  MoveL 1864 to (-16.69, 20.93, 85) mm, rotated rx 180 ry 0 rz -180 deg; joints [-156.025, -53.771, -94.051, 27.718, 60.883, -14.341]
  Call Extruder(17898.90608)
  MoveL 1865 to (-20.93, 16.69, 85) mm, rotated rx -180 ry 0 rz -180 deg; joints [-156.374, -53.467, -95.005, 27.167, 61.375, -13.813]
  Call Extruder(17908.27099)
  MoveL 1866 to (-24.11, 11.61, 85) mm, rotated rx -180 ry 0 rz 180 deg; joints [-156.928, -53.206, -95.842, 26.413, 61.758, -13.226]
  Call Extruder(17917.63579)
  MoveL 1867 to (-26.09, 5.96, 85) mm, rotated rx -180 ry 0 rz -180 deg; joints [-157.665, -52.998, -96.517, 25.49, 62.014, -12.61]
  Call Extruder(17927.00089)
  MoveL 1868 to (-26.77, 0, 85) mm, rotated rx 180 ry 0 rz -180 deg; joints [-158.546, -52.854, -96.993, 24.441, 62.127, -11.995]
  Call Extruder(17931.78963)
  MoveL 1869 to (-26.42, -3.05, 85) mm, rotated rx 180 ry 0 rz -180 deg; joints [-159.044, -52.814, -97.124, 23.87, 62.108, -11.695]
  Set speed (130.0 mm/s)
  MoveL 1870 to (-41.86, -6.3, 85) mm, rotated rx -180 ry 0 rz 180 deg; joints [-158.606, -52.066, -99.698, 23.975, 63.864, -11.084]
  Call Extruder(17936.78748)
  Set speed (60.0 mm/s)
  MoveL 1871 to (-41.51, -9.47, 85) mm, rotated rx -180 ry 0 rz 180 deg; joints [-159.151, -52.029, -99.83, 23.359, 63.847, -10.778]
  Call Extruder(17951.68313)
  MoveL 1872 to (-38.36, -18.47, 85) mm, rotated rx 180 ry 0 rz 180 deg; joints [-160.835, -52.023, -99.85, 21.508, 63.558, -9.953]
  Call Extruder(17966.57898)
  MoveL 1873 to (-33.28, -26.54, 85) mm, rotated rx 180 ry 0 rz 180 deg; joints [-162.466, -52.128, -99.478, 19.757, 63.035, -9.25]
  Call Extruder(17981.47480)
  MoveL 1874 to (-26.54, -33.28, 85) mm, rotated rx 180 ry 0 rz -180 deg; joints [-163.93, -52.339, -98.738, 18.218, 62.307, -8.696]
  Call Extruder(17996.37065)
  MoveL 1875 to (-18.47, -38.36, 85) mm, rotated rx 180 ry 0 rz 180 deg; joints [-165.137, -52.65, -97.673, 16.986, 61.41, -8.316]
  Call Extruder(18011.26630)
  MoveL 1876 to (-9.47, -41.51, 85) mm, rotated rx -180 ry 0 rz 180 deg; joints [-166.024, -53.05, -96.347, 16.127, 60.395, -8.129]
  Call Extruder(18026.16218)
  MoveL 1877 to (0, -42.57, 85) mm, rotated rx -180 ry 0 rz 180 deg; joints [-166.562, -53.521, -94.833, 15.678, 59.317, -8.151]
  Call Extruder(18033.93795)
  MoveL 1878 to (4.95, -42.02, 85) mm, rotated rx 180 ry 0 rz 180 deg; joints [-166.659, -53.791, -93.99, 15.659, 58.75, -8.274]
  Call Extruder(18041.05804)
  MoveL 1879 to (9.47, -41.51, 85) mm, rotated rx -180 ry 0 rz 180 deg; joints [-166.745, -54.043, -93.212, 15.646, 58.231, -8.388]
  Call Extruder(18055.95371)
  MoveL 1880 to (18.47, -38.36, 85) mm, rotated rx -180 ry 0 rz 180 deg; joints [-166.591, -54.589, -91.565, 16.015, 57.195, -8.839]
  Call Extruder(18070.84955)
  MoveL 1881 to (26.54, -33.29, 85) mm, rotated rx 180 ry 0 rz 180 deg; joints [-166.133, -55.132, -89.973, 16.751, 56.262, -9.49]
  Call Extruder(18085.74538)
  MoveL 1882 to (33.29, -26.54, 85) mm, rotated rx 180 ry 0 rz 180 deg; joints [-165.409, -55.642, -88.512, 17.803, 55.478, -10.315]
  Call Extruder(18100.64123)
  MoveL 1883 to (38.36, -18.47, 85) mm, rotated rx -180 ry 0 rz 180 deg; joints [-164.468, -56.091, -87.25, 19.109, 54.883, -11.272]
  Call Extruder(18115.53688)
  MoveL 1884 to (41.5, -9.47, 85) mm, rotated rx 180 ry 0 rz 180 deg; joints [-163.355, -56.454, -86.244, 20.599, 54.506, -12.31]
  Call Extruder(18130.43275)
  MoveL 1885 to (42.57, 0, 85) mm, rotated rx 180 ry 0 rz 180 deg; joints [-162.12, -56.711, -85.541, 22.195, 54.365, -13.372]
  Call Extruder(18145.32862)
  MoveL 1886 to (41.51, 9.47, 85) mm, rotated rx -180 ry 0 rz 180 deg; joints [-160.81, -56.847, -85.172, 23.824, 54.464, -14.393]
  Call Extruder(18160.22429)
  MoveL 1887 to (38.36, 18.47, 85) mm, rotated rx 180 ry 0 rz 180 deg; joints [-159.475, -56.853, -85.155, 25.41, 54.797, -15.316]
  Call Extruder(18175.12013)
  MoveL 1888 to (33.29, 26.54, 85) mm, rotated rx 180 ry 0 rz 180 deg; joints [-158.16, -56.73, -85.489, 26.888, 55.342, -16.085]
  Call Extruder(18190.01595)
  MoveL 1889 to (26.54, 33.28, 85) mm, rotated rx 180 ry 0 rz 180 deg; joints [-156.916, -56.485, -86.16, 28.2, 56.071, -16.662]
  Call Extruder(18204.91180)
  MoveL 1890 to (18.47, 38.36, 85) mm, rotated rx 180 ry 0 rz -180 deg; joints [-155.789, -56.131, -87.138, 29.294, 56.944, -17.016]
  Call Extruder(18219.80746)
  MoveL 1891 to (9.47, 41.51, 85) mm, rotated rx 180 ry 0 rz 180 deg; joints [-154.828, -55.689, -88.377, 30.132, 57.919, -17.133]
  Call Extruder(18234.70334)
  MoveL 1892 to (0, 42.57, 85) mm, rotated rx 180 ry 0 rz 180 deg; joints [-154.081, -55.184, -89.821, 30.678, 58.948, -17.014]
  Call Extruder(18249.59921)
  MoveL 1893 to (-9.47, 41.51, 85) mm, rotated rx 180 ry 0 rz 180 deg; joints [-153.594, -54.644, -91.403, 30.905, 59.984, -16.67]
  Call Extruder(18264.49486)
  MoveL 1894 to (-18.47, 38.36, 85) mm, rotated rx 180 ry 0 rz -180 deg; joints [-153.408, -54.096, -93.048, 30.791, 60.979, -16.124]
  Call Extruder(18279.39071)
  MoveL 1895 to (-26.54, 33.29, 85) mm, rotated rx 180 ry 0 rz 180 deg; joints [-153.557, -53.571, -94.676, 30.322, 61.888, -15.408]
  Call Extruder(18294.28653)
  MoveL 1896 to (-33.28, 26.54, 85) mm, rotated rx 180 ry 0 rz 180 deg; joints [-154.059, -53.094, -96.204, 29.499, 62.669, -14.561]
  Call Extruder(18309.18238)
  MoveL 1897 to (-38.36, 18.47, 85) mm, rotated rx 180 ry 0 rz -180 deg; joints [-154.913, -52.686, -97.552, 28.338, 63.284, -13.628]
  Call Extruder(18324.07804)
  MoveL 1898 to (-41.5, 9.47, 85) mm, rotated rx -180 ry 0 rz 180 deg; joints [-156.091, -52.366, -98.646, 26.877, 63.701, -12.656]
  Call Extruder(18338.97391)
  MoveL 1899 to (-42.57, 0, 85) mm, rotated rx 180 ry 0 rz -180 deg; joints [-157.533, -52.144, -99.421, 25.187, 63.894, -11.692]
  Call Extruder(18346.52819)
  MoveL 1900 to (-42.03, -4.8, 85) mm, rotated rx 180 ry 0 rz 180 deg; joints [-158.35, -52.084, -99.634, 24.263, 63.871, -11.227]
  Set speed (130.0 mm/s)
  MoveL 1901 to (-54.1, -7.67, 85) mm, rotated rx 180 ry 0 rz 180 deg; joints [-158.024, -51.54, -101.626, 24.334, 65.254, -10.72]
  Call Extruder(18350.60082)
  Set speed (30.0 mm/s)
  MoveL 1902 to (-53.59, -12.23, 85) mm, rotated rx 180 ry 0 rz -180 deg; joints [-158.835, -51.49, -101.819, 23.429, 65.236, -10.288]
  Call Extruder(18361.53095)
  MoveL 1903 to (-49.52, -23.85, 85) mm, rotated rx 180 ry 0 rz 180 deg; joints [-161.095, -51.483, -101.845, 20.97, 64.87, -9.244]
  Call Extruder(18372.46124)
  MoveL 1904 to (-42.98, -34.27, 85) mm, rotated rx -180 ry 0 rz 180 deg; joints [-163.275, -51.612, -101.354, 18.642, 64.197, -8.354]
  Call Extruder(18383.39136)
  MoveL 1905 to (-34.27, -42.98, 85) mm, rotated rx 180 ry 0 rz 180 deg; joints [-165.21, -51.876, -100.38, 16.611, 63.25, -7.647]
  Call Extruder(18394.32164)
  MoveL 1906 to (-23.85, -49.53, 85) mm, rotated rx 180 ry 0 rz 180 deg; joints [-166.774, -52.268, -98.985, 15.006, 62.083, -7.154]
  Call Extruder(18405.25177)
  MoveL 1907 to (-12.23, -53.59, 85) mm, rotated rx -180 ry 0 rz 180 deg; joints [-167.889, -52.775, -97.254, 13.913, 60.762, -6.899]
  Call Extruder(18416.18200)
  MoveL 1908 to (0, -54.97, 85) mm, rotated rx -180 ry 0 rz 180 deg; joints [-168.526, -53.378, -95.288, 13.367, 59.36, -6.905]
  Call Extruder(18421.83349)
  MoveL 1909 to (6.32, -54.26, 85) mm, rotated rx 180 ry 0 rz 180 deg; joints [-168.616, -53.721, -94.208, 13.366, 58.632, -7.051]
  Call Extruder(18427.11222)
  MoveL 1910 to (12.23, -53.59, 85) mm, rotated rx -180 ry 0 rz 180 deg; joints [-168.697, -54.05, -93.19, 13.37, 57.952, -7.188]
  Call Extruder(18438.04236)
  MoveL 1911 to (23.85, -49.53, 85) mm, rotated rx 180 ry 0 rz 180 deg; joints [-168.436, -54.757, -91.068, 13.891, 56.611, -7.75]
  Call Extruder(18448.97264)
  MoveL 1912 to (34.27, -42.98, 85) mm, rotated rx 180 ry 0 rz 180 deg; joints [-167.797, -55.462, -89.022, 14.879, 55.403, -8.579]
  Call Extruder(18459.90276)
  MoveL 1913 to (42.98, -34.27, 85) mm, rotated rx -180 ry 0 rz 180 deg; joints [-166.837, -56.127, -87.148, 16.266, 54.391, -9.642]
  Call Extruder(18470.83304)
  MoveL 1914 to (49.53, -23.85, 85) mm, rotated rx -180 ry 0 rz 180 deg; joints [-165.618, -56.714, -85.531, 17.968, 53.624, -10.888]
  Call Extruder(18481.76317)
  MoveL 1915 to (53.59, -12.23, 85) mm, rotated rx 180 ry 0 rz -180 deg; joints [-164.2, -57.19, -84.244, 19.895, 53.141, -12.248]
  Call Extruder(18492.69340)
  MoveL 1916 to (54.97, 0, 85) mm, rotated rx 180 ry 0 rz 180 deg; joints [-162.641, -57.527, -83.344, 21.948, 52.964, -13.643]
  Call Extruder(18503.62362)
  MoveL 1917 to (53.59, 12.23, 85) mm, rotated rx 180 ry 0 rz 180 deg; joints [-160.996, -57.705, -82.872, 24.029, 53.1, -14.986]
  Call Extruder(18514.55376)
  MoveL 1918 to (49.52, 23.85, 85) mm, rotated rx -180 ry 0 rz -180 deg; joints [-159.322, -57.714, -82.85, 26.044, 53.537, -16.195]
  Call Extruder(18525.48404)
  MoveL 1919 to (42.98, 34.27, 85) mm, rotated rx -180 ry 0 rz 180 deg; joints [-157.673, -57.552, -83.278, 27.912, 54.249, -17.198]
  Call Extruder(18536.41416)
  MoveL 1920 to (34.27, 42.98, 85) mm, rotated rx -180 ry 0 rz 180 deg; joints [-156.102, -57.23, -84.137, 29.563, 55.194, -17.94]
  Call Extruder(18547.34444)
  MoveL 1921 to (23.85, 49.52, 85) mm, rotated rx -180 ry 0 rz 180 deg; joints [-154.667, -56.767, -85.388, 30.942, 56.322, -18.388]
  Call Extruder(18558.27458)
  MoveL 1922 to (12.23, 53.59, 85) mm, rotated rx 180 ry 0 rz 180 deg; joints [-153.426, -56.19, -86.975, 32.004, 57.576, -18.526]
  Call Extruder(18569.20480)
  MoveL 1923 to (0, 54.97, 85) mm, rotated rx -180 ry 0 rz 180 deg; joints [-152.438, -55.531, -88.827, 32.711, 58.896, -18.355]
  Call Extruder(18580.13502)
  MoveL 1924 to (-12.23, 53.59, 85) mm, rotated rx 180 ry 0 rz 180 deg; joints [-151.764, -54.828, -90.86, 33.03, 60.223, -17.894]
  Call Extruder(18591.06516)
  MoveL 1925 to (-23.85, 49.52, 85) mm, rotated rx 180 ry 0 rz 180 deg; joints [-151.463, -54.119, -92.979, 32.93, 61.497, -17.175]
  Call Extruder(18601.99544)
  MoveL 1926 to (-34.27, 42.98, 85) mm, rotated rx 180 ry 0 rz 180 deg; joints [-151.589, -53.442, -95.084, 32.385, 62.663, -16.239]
  Call Extruder(18612.92556)
  MoveL 1927 to (-42.98, 34.27, 85) mm, rotated rx 180 ry 0 rz -180 deg; joints [-152.179, -52.831, -97.068, 31.381, 63.669, -15.139]
  Call Extruder(18623.85584)
  MoveL 1928 to (-49.52, 23.85, 85) mm, rotated rx 180 ry 0 rz 180 deg; joints [-153.248, -52.313, -98.827, 29.924, 64.469, -13.933]
  Call Extruder(18634.78598)
  MoveL 1929 to (-53.59, 12.23, 85) mm, rotated rx 180 ry 0 rz 180 deg; joints [-154.769, -51.91, -100.259, 28.051, 65.018, -12.683]
  Call Extruder(18645.71620)
  MoveL 1930 to (-54.97, 0, 85) mm, rotated rx 180 ry 0 rz -180 deg; joints [-156.673, -51.633, -101.278, 25.844, 65.282, -11.45]
  Call Extruder(18651.24182)
  MoveL 1931 to (-54.27, -6.18, 85) mm, rotated rx 180 ry 0 rz -180 deg; joints [-157.76, -51.558, -101.561, 24.629, 65.26, -10.861]
  Set speed (130.0 mm/s)
  MoveL 1932 to (-49.9, -9.51, 85) mm, rotated rx -180 ry 0 rz 180 deg; joints [-158.616, -51.679, -101.105, 23.764, 64.795, -10.62]
  MoveL 1933 to (1.69, -13.14, 85) mm, rotated rx 180 ry 0 rz -180 deg; joints [-162.112, -54.05, -93.191, 20.997, 59.006, -11.18]
  Call Extruder(18653.24626)
  Set speed (80.0 mm/s)
  MoveL 1934 to (2.97, -12.99, 85) mm, rotated rx -180 ry 0 rz -180 deg; joints [-162.152, -54.121, -92.974, 20.982, 58.862, -11.217]
  Call Extruder(18657.90984)
  MoveL 1935 to (5.78, -12.01, 85) mm, rotated rx 180 ry 0 rz -180 deg; joints [-162.141, -54.291, -92.457, 21.071, 58.541, -11.37]
  Call Extruder(18662.57346)
  MoveL 1936 to (8.31, -10.42, 85) mm, rotated rx -180 ry 0 rz -180 deg; joints [-162.027, -54.459, -91.954, 21.277, 58.25, -11.581]
  Call Extruder(18667.23766)
  MoveL 1937 to (10.42, -8.31, 85) mm, rotated rx 180 ry 0 rz -180 deg; joints [-161.819, -54.615, -91.489, 21.587, 58.005, -11.84]
  Call Extruder(18671.90129)
  MoveL 1938 to (12.01, -5.78, 85) mm, rotated rx -180 ry 0 rz 180 deg; joints [-161.529, -54.751, -91.086, 21.984, 57.817, -12.135]
  Call Extruder(18676.56485)
  MoveL 1939 to (12.99, -2.97, 85) mm, rotated rx -180 ry 0 rz -180 deg; joints [-161.171, -54.861, -90.763, 22.448, 57.696, -12.451]
  Call Extruder(18681.22881)
  MoveL 1940 to (13.33, 0, 85) mm, rotated rx 180 ry 0 rz -180 deg; joints [-160.763, -54.938, -90.537, 22.956, 57.648, -12.771]
  Call Extruder(18685.89276)
  MoveL 1941 to (12.99, 2.97, 85) mm, rotated rx 180 ry 0 rz 180 deg; joints [-160.324, -54.979, -90.418, 23.482, 57.674, -13.078]
  Call Extruder(18690.55633)
  MoveL 1942 to (12.01, 5.78, 85) mm, rotated rx -180 ry 0 rz -180 deg; joints [-159.874, -54.981, -90.412, 24.001, 57.774, -13.357]
  Call Extruder(18695.21996)
  MoveL 1943 to (10.42, 8.31, 85) mm, rotated rx -180 ry 0 rz 180 deg; joints [-159.432, -54.944, -90.52, 24.489, 57.941, -13.592]
  Call Extruder(18699.88415)
  MoveL 1944 to (8.31, 10.42, 85) mm, rotated rx 180 ry 0 rz 180 deg; joints [-159.021, -54.87, -90.736, 24.924, 58.168, -13.771]
  Call Extruder(18704.54778)
  MoveL 1945 to (5.78, 12.01, 85) mm, rotated rx 180 ry 0 rz -180 deg; joints [-158.657, -54.763, -91.05, 25.285, 58.442, -13.886]
  Call Extruder(18709.21134)
  MoveL 1946 to (2.97, 12.99, 85) mm, rotated rx -180 ry 0 rz 180 deg; joints [-158.359, -54.629, -91.446, 25.555, 58.75, -13.931]
  Call Extruder(18713.87530)
  MoveL 1947 to (0, 13.33, 85) mm, rotated rx 180 ry 0 rz 180 deg; joints [-158.143, -54.475, -91.906, 25.72, 59.078, -13.903]
  Call Extruder(18718.53925)
  MoveL 1948 to (-2.97, 13, 85) mm, rotated rx 180 ry 0 rz 180 deg; joints [-158.019, -54.308, -92.406, 25.774, 59.408, -13.806]
  Call Extruder(18723.20282)
  MoveL 1949 to (-5.78, 12.01, 85) mm, rotated rx 180 ry 0 rz 180 deg; joints [-157.997, -54.138, -92.923, 25.71, 59.725, -13.644]
  Call Extruder(18727.86645)
  MoveL 1950 to (-8.31, 10.42, 85) mm, rotated rx 180 ry 0 rz 180 deg; joints [-158.08, -53.972, -93.43, 25.531, 60.013, -13.427]
  Call Extruder(18732.53064)
  MoveL 1951 to (-10.42, 8.31, 85) mm, rotated rx 180 ry 0 rz 180 deg; joints [-158.266, -53.819, -93.901, 25.244, 60.259, -13.165]
  Call Extruder(18737.19427)
  MoveL 1952 to (-12.01, 5.78, 85) mm, rotated rx -180 ry 0 rz 180 deg; joints [-158.549, -53.687, -94.314, 24.86, 60.448, -12.872]
  Call Extruder(18741.85784)
  MoveL 1953 to (-12.99, 2.97, 85) mm, rotated rx -180 ry 0 rz -180 deg; joints [-158.913, -53.581, -94.645, 24.398, 60.573, -12.563]
  Call Extruder(18746.52180)
  MoveL 1954 to (-13.33, 0, 85) mm, rotated rx 180 ry 0 rz 180 deg; joints [-159.341, -53.507, -94.878, 23.881, 60.627, -12.253]
  Call Extruder(18751.18574)
  MoveL 1955 to (-12.99, -2.97, 85) mm, rotated rx 180 ry 0 rz 180 deg; joints [-159.811, -53.468, -95.001, 23.336, 60.605, -11.956]
  Call Extruder(18755.84931)
  MoveL 1956 to (-12.01, -5.78, 85) mm, rotated rx 180 ry 0 rz 180 deg; joints [-160.294, -53.467, -95.007, 22.791, 60.51, -11.687]
  Call Extruder(18760.51294)
  MoveL 1957 to (-10.42, -8.31, 85) mm, rotated rx 180 ry 0 rz 180 deg; joints [-160.766, -53.502, -94.895, 22.276, 60.345, -11.458]
  Call Extruder(18765.17714)
  MoveL 1958 to (-8.31, -10.42, 85) mm, rotated rx -180 ry 0 rz 180 deg; joints [-161.2, -53.572, -94.673, 21.819, 60.118, -11.281]
  Call Extruder(18769.84076)
  MoveL 1959 to (-5.78, -12.01, 85) mm, rotated rx 180 ry 0 rz 180 deg; joints [-161.572, -53.675, -94.35, 21.445, 59.842, -11.163]
  Call Extruder(18774.50433)
  MoveL 1960 to (-2.97, -12.99, 85) mm, rotated rx 180 ry 0 rz 180 deg; joints [-161.863, -53.805, -93.945, 21.173, 59.529, -11.112]
  Call Extruder(18779.16829)
  MoveL 1961 to (0, -13.33, 85) mm, rotated rx -180 ry 0 rz -180 deg; joints [-162.059, -53.956, -93.479, 21.016, 59.197, -11.13]
  Call Extruder(18781.82779)
  MoveL 1962 to (1.69, -13.14, 85) mm, rotated rx 180 ry 0 rz -180 deg; joints [-162.112, -54.05, -93.191, 20.997, 59.006, -11.18]
  Set speed (130.0 mm/s)
  MoveL 1963 to (1.69, -13.14, 90) mm, rotated rx -180 ry 0 rz -180 deg; joints [-162.112, -53.285, -93.531, 21.089, 58.609, -11.358]
  MoveL 1964 to (-26.25, -4.54, 90) mm, rotated rx 180 ry 0 rz 180 deg; joints [-159.288, -52.001, -97.533, 23.686, 61.689, -11.752]
  Call Extruder(18784.06040)
  Set speed (60.0 mm/s)
  MoveL 1965 to (-26.09, -5.96, 90) mm, rotated rx 180 ry 0 rz 180 deg; joints [-159.522, -51.983, -97.591, 23.417, 61.678, -11.611]
  Call Extruder(18793.42519)
  MoveL 1966 to (-24.11, -11.61, 90) mm, rotated rx 180 ry 0 rz 180 deg; joints [-160.532, -51.979, -97.604, 22.29, 61.488, -11.072]
  Call Extruder(18802.79012)
  MoveL 1967 to (-20.93, -16.69, 90) mm, rotated rx 180 ry 0 rz -180 deg; joints [-161.513, -52.049, -97.375, 21.223, 61.156, -10.611]
  Call Extruder(18812.15532)
  MoveL 1968 to (-16.69, -20.93, 90) mm, rotated rx -180 ry 0 rz 180 deg; joints [-162.406, -52.191, -96.919, 20.28, 60.7, -10.25]
  Call Extruder(18821.52024)
  MoveL 1969 to (-11.61, -24.12, 90) mm, rotated rx 180 ry 0 rz 180 deg; joints [-163.159, -52.398, -96.261, 19.515, 60.143, -10.006]
  Call Extruder(18830.88503)
  MoveL 1970 to (-5.96, -26.09, 90) mm, rotated rx 180 ry 0 rz 180 deg; joints [-163.733, -52.66, -95.437, 18.968, 59.514, -9.891]
  Call Extruder(18840.25014)
  MoveL 1971 to (0, -26.77, 90) mm, rotated rx -180 ry 0 rz 180 deg; joints [-164.103, -52.968, -94.491, 18.667, 58.846, -9.914]
  Call Extruder(18845.91642)
  MoveL 1972 to (3.6, -26.36, 90) mm, rotated rx 180 ry 0 rz 180 deg; joints [-164.198, -53.17, -93.876, 18.638, 58.439, -10.012]
  Call Extruder(18849.61524)
  MoveL 1973 to (5.96, -26.09, 90) mm, rotated rx 180 ry 0 rz 180 deg; joints [-164.258, -53.304, -93.473, 18.622, 58.173, -10.076]
  Call Extruder(18858.98004)
  MoveL 1974 to (11.61, -24.11, 90) mm, rotated rx -180 ry 0 rz 180 deg; joints [-164.201, -53.654, -92.434, 18.827, 57.531, -10.373]
  Call Extruder(18868.34495)
  MoveL 1975 to (16.69, -20.93, 90) mm, rotated rx -180 ry 0 rz 180 deg; joints [-163.944, -53.999, -91.426, 19.267, 56.952, -10.792]
  Call Extruder(18877.71016)
  MoveL 1976 to (20.93, -16.69, 90) mm, rotated rx 180 ry 0 rz 180 deg; joints [-163.508, -54.322, -90.498, 19.912, 56.466, -11.316]
  Call Extruder(18887.07508)
  MoveL 1977 to (24.11, -11.61, 90) mm, rotated rx -180 ry 0 rz 180 deg; joints [-162.92, -54.605, -89.695, 20.725, 56.096, -11.918]
  Call Extruder(18896.43987)
  MoveL 1978 to (26.09, -5.96, 90) mm, rotated rx -180 ry 0 rz -180 deg; joints [-162.209, -54.833, -89.054, 21.663, 55.862, -12.566]
  Call Extruder(18905.80498)
  MoveL 1979 to (26.77, 0, 90) mm, rotated rx 180 ry 0 rz -180 deg; joints [-161.41, -54.994, -88.605, 22.679, 55.773, -13.227]
  Call Extruder(18915.17008)
  MoveL 1980 to (26.09, 5.96, 90) mm, rotated rx 180 ry 0 rz 180 deg; joints [-160.556, -55.079, -88.37, 23.723, 55.835, -13.863]
  Call Extruder(18924.53488)
  MoveL 1981 to (24.12, 11.61, 90) mm, rotated rx 180 ry 0 rz 180 deg; joints [-159.683, -55.083, -88.359, 24.747, 56.042, -14.439]
  Call Extruder(18933.89980)
  MoveL 1982 to (20.93, 16.69, 90) mm, rotated rx -180 ry 0 rz 180 deg; joints [-158.826, -55.006, -88.572, 25.706, 56.383, -14.924]
  Call Extruder(18943.26501)
  MoveL 1983 to (16.69, 20.93, 90) mm, rotated rx 180 ry 0 rz 180 deg; joints [-158.019, -54.852, -89.001, 26.558, 56.839, -15.292]
  Call Extruder(18952.62991)
  MoveL 1984 to (11.61, 24.11, 90) mm, rotated rx 180 ry 0 rz 180 deg; joints [-157.299, -54.63, -89.624, 27.268, 57.389, -15.525]
  Call Extruder(18961.99472)
  MoveL 1985 to (5.96, 26.09, 90) mm, rotated rx -180 ry 0 rz 180 deg; joints [-156.697, -54.352, -90.413, 27.805, 58.003, -15.612]
  Call Extruder(18971.35983)
  MoveL 1986 to (0, 26.77, 90) mm, rotated rx 180 ry 0 rz 180 deg; joints [-156.245, -54.033, -91.33, 28.144, 58.652, -15.551]
  Call Extruder(18980.72493)
  MoveL 1987 to (-5.96, 26.09, 90) mm, rotated rx 180 ry 0 rz 180 deg; joints [-155.969, -53.689, -92.332, 28.267, 59.306, -15.348]
  Call Extruder(18990.08972)
  MoveL 1988 to (-11.61, 24.12, 90) mm, rotated rx 180 ry 0 rz 180 deg; joints [-155.891, -53.339, -93.37, 28.163, 59.932, -15.015]
  Call Extruder(18999.45464)
  MoveL 1989 to (-16.69, 20.93, 90) mm, rotated rx 180 ry 0 rz -180 deg; joints [-156.025, -53, -94.392, 27.83, 60.502, -14.571]
  Call Extruder(19008.81985)
  MoveL 1990 to (-20.93, 16.69, 90) mm, rotated rx 180 ry 0 rz 180 deg; joints [-156.374, -52.689, -95.348, 27.276, 60.987, -14.04]
  Call Extruder(19018.18476)
  MoveL 1991 to (-24.11, 11.61, 90) mm, rotated rx -180 ry 0 rz 180 deg; joints [-156.928, -52.421, -96.186, 26.519, 61.364, -13.449]
  Call Extruder(19027.54956)
  MoveL 1992 to (-26.09, 5.96, 90) mm, rotated rx 180 ry 0 rz 180 deg; joints [-157.665, -52.209, -96.862, 25.592, 61.613, -12.828]
  Call Extruder(19036.91467)
  MoveL 1993 to (-26.77, 0, 90) mm, rotated rx 180 ry 0 rz 180 deg; joints [-158.546, -52.06, -97.34, 24.539, 61.721, -12.205]
  Call Extruder(19041.70340)
  MoveL 1994 to (-26.42, -3.05, 90) mm, rotated rx 180 ry 0 rz -180 deg; joints [-159.044, -52.02, -97.471, 23.967, 61.699, -11.901]
  Set speed (130.0 mm/s)
  MoveL 1995 to (-41.86, -6.3, 90) mm, rotated rx 180 ry 0 rz 180 deg; joints [-158.606, -51.249, -100.051, 24.068, 63.44, -11.294]
  Call Extruder(19046.70125)
  Set speed (60.0 mm/s)
  MoveL 1996 to (-41.5, -9.47, 90) mm, rotated rx 180 ry 0 rz 180 deg; joints [-159.151, -51.211, -100.184, 23.45, 63.422, -10.984]
  Call Extruder(19061.59690)
  MoveL 1997 to (-38.36, -18.47, 90) mm, rotated rx -180 ry 0 rz 180 deg; joints [-160.835, -51.205, -100.203, 21.594, 63.126, -10.144]
  Call Extruder(19076.49275)
  MoveL 1998 to (-33.29, -26.54, 90) mm, rotated rx -180 ry 0 rz 180 deg; joints [-162.466, -51.313, -99.831, 19.837, 62.601, -9.426]
  Call Extruder(19091.38857)
  MoveL 1999 to (-26.54, -33.28, 90) mm, rotated rx 180 ry 0 rz -180 deg; joints [-163.93, -51.531, -99.088, 18.294, 61.872, -8.859]
  Call Extruder(19106.28442)
  MoveL 2000 to (-18.47, -38.36, 90) mm, rotated rx -180 ry 0 rz 180 deg; joints [-165.137, -51.851, -98.022, 17.058, 60.979, -8.467]
  Call Extruder(19121.18007)
  MoveL 2001 to (-9.47, -41.5, 90) mm, rotated rx 180 ry 0 rz 180 deg; joints [-166.024, -52.262, -96.692, 16.198, 59.97, -8.272]
  Call Extruder(19136.07595)
  MoveL 2002 to (0, -42.57, 90) mm, rotated rx -180 ry 0 rz 180 deg; joints [-166.562, -52.745, -95.176, 15.748, 58.898, -8.288]
  Call Extruder(19144.50777)
  MoveL 2003 to (5.36, -41.97, 90) mm, rotated rx 180 ry 0 rz -180 deg; joints [-166.667, -53.044, -94.259, 15.729, 58.288, -8.421]
  Call Extruder(19150.97182)
  MoveL 2004 to (9.47, -41.51, 90) mm, rotated rx -180 ry 0 rz 180 deg; joints [-166.745, -53.278, -93.551, 15.718, 57.821, -8.524]
  Call Extruder(19165.86748)
  MoveL 2005 to (18.47, -38.36, 90) mm, rotated rx -180 ry 0 rz 180 deg; joints [-166.591, -53.836, -91.901, 16.09, 56.795, -8.977]
  Call Extruder(19180.76333)
  MoveL 2006 to (26.54, -33.29, 90) mm, rotated rx 180 ry 0 rz 180 deg; joints [-166.133, -54.389, -90.308, 16.831, 55.871, -9.633]
  Call Extruder(19195.65915)
  MoveL 2007 to (33.29, -26.54, 90) mm, rotated rx -180 ry 0 rz 180 deg; joints [-165.409, -54.908, -88.845, 17.889, 55.096, -10.464]
  Call Extruder(19210.55500)
  MoveL 2008 to (38.36, -18.47, 90) mm, rotated rx 180 ry 0 rz 180 deg; joints [-164.468, -55.365, -87.581, 19.201, 54.51, -11.43]
  Call Extruder(19225.45065)
  MoveL 2009 to (41.51, -9.47, 90) mm, rotated rx 180 ry 0 rz 180 deg; joints [-163.355, -55.734, -86.575, 20.697, 54.141, -12.48]
  Call Extruder(19240.34652)
  MoveL 2010 to (42.57, 0, 90) mm, rotated rx 180 ry 0 rz 180 deg; joints [-162.12, -55.995, -85.871, 22.301, 54.007, -13.552]
  Call Extruder(19255.24240)
  MoveL 2011 to (41.51, 9.47, 90) mm, rotated rx -180 ry 0 rz -180 deg; joints [-160.81, -56.132, -85.502, 23.936, 54.113, -14.585]
  Call Extruder(19270.13806)
  MoveL 2012 to (38.36, 18.47, 90) mm, rotated rx 180 ry 0 rz 180 deg; joints [-159.475, -56.139, -85.484, 25.528, 54.449, -15.518]
  Call Extruder(19285.03390)
  MoveL 2013 to (33.29, 26.54, 90) mm, rotated rx 180 ry 0 rz 180 deg; joints [-158.16, -56.014, -85.819, 27.01, 54.998, -16.299]
  Call Extruder(19299.92973)
  MoveL 2014 to (26.54, 33.28, 90) mm, rotated rx -180 ry 0 rz 180 deg; joints [-156.916, -55.765, -86.491, 28.324, 55.728, -16.884]
  Call Extruder(19314.82557)
  MoveL 2015 to (18.47, 38.36, 90) mm, rotated rx -180 ry 0 rz -180 deg; joints [-155.789, -55.406, -87.469, 29.421, 56.601, -17.247]
  Call Extruder(19329.72123)
  MoveL 2016 to (9.47, 41.51, 90) mm, rotated rx -180 ry 0 rz 180 deg; joints [-154.828, -54.956, -88.71, 30.259, 57.573, -17.371]
  Call Extruder(19344.61711)
  MoveL 2017 to (0, 42.57, 90) mm, rotated rx 180 ry 0 rz 180 deg; joints [-154.081, -54.442, -90.155, 30.804, 58.598, -17.258]
  Call Extruder(19359.51298)
  MoveL 2018 to (-9.47, 41.51, 90) mm, rotated rx -180 ry 0 rz 180 deg; joints [-153.594, -53.891, -91.74, 31.029, 59.627, -16.918]
  Call Extruder(19374.40863)
  MoveL 2019 to (-18.47, 38.36, 90) mm, rotated rx 180 ry 0 rz 180 deg; joints [-153.408, -53.333, -93.387, 30.912, 60.614, -16.373]
  Call Extruder(19389.30448)
  MoveL 2020 to (-26.54, 33.29, 90) mm, rotated rx -180 ry 0 rz 180 deg; joints [-153.557, -52.796, -95.018, 30.441, 61.514, -15.657]
  Call Extruder(19404.20030)
  MoveL 2021 to (-33.28, 26.54, 90) mm, rotated rx 180 ry 0 rz 180 deg; joints [-154.059, -52.307, -96.549, 29.613, 62.284, -14.807]
  Call Extruder(19419.09615)
  MoveL 2022 to (-38.36, 18.47, 90) mm, rotated rx -180 ry 0 rz 180 deg; joints [-154.913, -51.888, -97.9, 28.446, 62.888, -13.868]
  Call Extruder(19433.99181)
  MoveL 2023 to (-41.5, 9.47, 90) mm, rotated rx -180 ry 0 rz 180 deg; joints [-156.091, -51.558, -98.996, 26.981, 63.294, -12.887]
  Call Extruder(19448.88768)
  MoveL 2024 to (-42.57, 0, 90) mm, rotated rx 180 ry 0 rz -180 deg; joints [-157.533, -51.33, -99.773, 25.284, 63.477, -11.911]
  Call Extruder(19456.44196)
  MoveL 2025 to (-42.03, -4.8, 90) mm, rotated rx 180 ry 0 rz 180 deg; joints [-158.35, -51.268, -99.987, 24.357, 63.449, -11.44]
  Set speed (130.0 mm/s)
  MoveL 2026 to (-54.1, -7.67, 90) mm, rotated rx 180 ry 0 rz 180 deg; joints [-158.024, -50.706, -101.985, 24.426, 64.821, -10.936]
  Call Extruder(19460.51459)
  Set speed (30.0 mm/s)
  MoveL 2027 to (-53.59, -12.23, 90) mm, rotated rx -180 ry 0 rz 180 deg; joints [-158.835, -50.654, -102.178, 23.518, 64.798, -10.498]
  Call Extruder(19471.44473)
  MoveL 2028 to (-49.52, -23.85, 90) mm, rotated rx 180 ry 0 rz 180 deg; joints [-161.095, -50.647, -102.204, 21.051, 64.425, -9.433]
  Call Extruder(19482.37501)
  MoveL 2029 to (-42.98, -34.27, 90) mm, rotated rx 180 ry 0 rz 180 deg; joints [-163.275, -50.781, -101.712, 18.716, 63.748, -8.523]
  Call Extruder(19493.30513)
  MoveL 2030 to (-34.27, -42.98, 90) mm, rotated rx -180 ry 0 rz 180 deg; joints [-165.21, -51.054, -100.735, 16.679, 62.802, -7.798]
  Call Extruder(19504.23541)
  MoveL 2031 to (-23.85, -49.53, 90) mm, rotated rx -180 ry 0 rz 180 deg; joints [-166.774, -51.458, -99.336, 15.07, 61.64, -7.289]
  Call Extruder(19515.16555)
  MoveL 2032 to (-12.23, -53.59, 90) mm, rotated rx 180 ry 0 rz 180 deg; joints [-167.889, -51.98, -97.602, 13.974, 60.327, -7.023]
  Call Extruder(19526.09577)
  MoveL 2033 to (0, -54.97, 90) mm, rotated rx -180 ry 0 rz 180 deg; joints [-168.526, -52.598, -95.631, 13.428, 58.935, -7.023]
  Call Extruder(19532.12010)
  MoveL 2034 to (6.74, -54.21, 90) mm, rotated rx 180 ry 0 rz 180 deg; joints [-168.622, -52.972, -94.477, 13.428, 58.165, -7.178]
  Call Extruder(19537.02599)
  MoveL 2035 to (12.23, -53.59, 90) mm, rotated rx 180 ry 0 rz 180 deg; joints [-168.697, -53.285, -93.529, 13.432, 57.539, -7.305]
  Call Extruder(19547.95613)
  MoveL 2036 to (23.85, -49.53, 90) mm, rotated rx 180 ry 0 rz 180 deg; joints [-168.436, -54.007, -91.404, 13.957, 56.209, -7.87]
  Call Extruder(19558.88641)
  MoveL 2037 to (34.27, -42.98, 90) mm, rotated rx -180 ry 0 rz 180 deg; joints [-167.797, -54.725, -89.355, 14.951, 55.013, -8.705]
  Call Extruder(19569.81653)
  MoveL 2038 to (42.98, -34.27, 90) mm, rotated rx -180 ry 0 rz 180 deg; joints [-166.837, -55.402, -87.48, 16.346, 54.012, -9.778]
  Call Extruder(19580.74681)
  MoveL 2039 to (49.53, -23.85, 90) mm, rotated rx 180 ry 0 rz 180 deg; joints [-165.618, -55.998, -85.861, 18.057, 53.256, -11.036]
  Call Extruder(19591.67695)
  MoveL 2040 to (53.59, -12.23, 90) mm, rotated rx 180 ry 0 rz -180 deg; joints [-164.2, -56.481, -84.573, 19.993, 52.783, -12.411]
  Call Extruder(19602.60717)
  MoveL 2041 to (54.97, 0, 90) mm, rotated rx 180 ry 0 rz 180 deg; joints [-162.641, -56.823, -83.672, 22.055, 52.615, -13.82]
  Call Extruder(19613.53739)
  MoveL 2042 to (53.59, 12.23, 90) mm, rotated rx -180 ry 0 rz 180 deg; joints [-160.996, -57.003, -83.2, 24.144, 52.758, -15.177]
  Call Extruder(19624.46753)
  MoveL 2043 to (49.52, 23.85, 90) mm, rotated rx 180 ry 0 rz -180 deg; joints [-159.322, -57.012, -83.178, 26.166, 53.201, -16.4]
  Call Extruder(19635.39781)
  MoveL 2044 to (42.98, 34.27, 90) mm, rotated rx 180 ry 0 rz 180 deg; joints [-157.673, -56.848, -83.606, 28.039, 53.917, -17.415]
  Call Extruder(19646.32793)
  MoveL 2045 to (34.27, 42.98, 90) mm, rotated rx 180 ry 0 rz 180 deg; joints [-156.102, -56.522, -84.465, 29.694, 54.863, -18.17]
  Call Extruder(19657.25821)
  MoveL 2046 to (23.85, 49.52, 90) mm, rotated rx 180 ry 0 rz 180 deg; joints [-154.667, -56.052, -85.717, 31.075, 55.991, -18.628]
  Call Extruder(19668.18835)
  MoveL 2047 to (12.23, 53.59, 90) mm, rotated rx -180 ry 0 rz 180 deg; joints [-153.426, -55.465, -87.306, 32.137, 57.242, -18.774]
  Call Extruder(19679.11857)
  MoveL 2048 to (0, 54.97, 90) mm, rotated rx 180 ry 0 rz 180 deg; joints [-152.438, -54.795, -89.16, 32.843, 58.558, -18.61]
  Call Extruder(19690.04880)
  MoveL 2049 to (-12.23, 53.59, 90) mm, rotated rx 180 ry 0 rz 180 deg; joints [-151.764, -54.079, -91.195, 33.16, 59.877, -18.155]
  Call Extruder(19700.97893)
  MoveL 2050 to (-23.85, 49.52, 90) mm, rotated rx 180 ry 0 rz 180 deg; joints [-151.463, -53.356, -93.318, 33.056, 61.141, -17.438]
  Call Extruder(19711.90921)
  MoveL 2051 to (-34.27, 42.98, 90) mm, rotated rx 180 ry 0 rz 180 deg; joints [-151.589, -52.664, -95.426, 32.507, 62.295, -16.503]
  Call Extruder(19722.83933)
  MoveL 2052 to (-42.98, 34.27, 90) mm, rotated rx 180 ry 0 rz -180 deg; joints [-152.179, -52.037, -97.415, 31.498, 63.287, -15.4]
  Call Extruder(19733.76961)
  MoveL 2053 to (-49.52, 23.85, 90) mm, rotated rx 180 ry 0 rz 180 deg; joints [-153.248, -51.505, -99.177, 30.034, 64.072, -14.187]
  Call Extruder(19744.69975)
  MoveL 2054 to (-53.59, 12.23, 90) mm, rotated rx 180 ry 0 rz 180 deg; joints [-154.769, -51.088, -100.613, 28.155, 64.606, -12.926]
  Call Extruder(19755.62998)
  MoveL 2055 to (-54.97, 0, 90) mm, rotated rx 180 ry 0 rz -180 deg; joints [-156.673, -50.802, -101.636, 25.94, 64.856, -11.678]
  Call Extruder(19761.15559)
  MoveL 2056 to (-54.27, -6.18, 90) mm, rotated rx 180 ry 0 rz -180 deg; joints [-157.76, -50.724, -101.919, 24.721, 64.828, -11.08]
  Set speed (130.0 mm/s)
  MoveL 2057 to (-49.9, -9.51, 90) mm, rotated rx -180 ry 0 rz 180 deg; joints [-158.616, -50.85, -101.462, 23.855, 64.363, -10.831]
  MoveL 2058 to (2.11, -13.09, 90) mm, rotated rx -180 ry 0 rz -180 deg; joints [-162.125, -53.309, -93.459, 21.084, 58.562, -11.37]
  Call Extruder(19762.50397)
  Set speed (80.0 mm/s)
  MoveL 2059 to (2.97, -12.99, 90) mm, rotated rx 180 ry 0 rz -180 deg; joints [-162.152, -53.358, -93.313, 21.075, 58.466, -11.395]
  Call Extruder(19767.16754)
  MoveL 2060 to (5.78, -12.01, 90) mm, rotated rx 180 ry 0 rz 180 deg; joints [-162.141, -53.532, -92.795, 21.165, 58.148, -11.548]
  Call Extruder(19771.83117)
  MoveL 2061 to (8.31, -10.42, 90) mm, rotated rx 180 ry 0 rz -180 deg; joints [-162.027, -53.703, -92.291, 21.372, 57.86, -11.76]
  Call Extruder(19776.49536)
  MoveL 2062 to (10.42, -8.31, 90) mm, rotated rx 180 ry 0 rz -180 deg; joints [-161.819, -53.862, -91.826, 21.683, 57.618, -12.021]
  Call Extruder(19781.15899)
  MoveL 2063 to (12.01, -5.78, 90) mm, rotated rx -180 ry 0 rz 180 deg; joints [-161.529, -54.001, -91.422, 22.083, 57.433, -12.319]
  Call Extruder(19785.82256)
  MoveL 2064 to (12.99, -2.97, 90) mm, rotated rx -180 ry 0 rz -180 deg; joints [-161.171, -54.113, -91.099, 22.549, 57.315, -12.638]
  Call Extruder(19790.48651)
  MoveL 2065 to (13.33, 0, 90) mm, rotated rx 180 ry 0 rz 180 deg; joints [-160.763, -54.191, -90.872, 23.058, 57.269, -12.961]
  Call Extruder(19795.15046)
  MoveL 2066 to (13, 2.97, 90) mm, rotated rx -180 ry 0 rz 180 deg; joints [-160.324, -54.233, -90.753, 23.586, 57.298, -13.273]
  Call Extruder(19799.81404)
  MoveL 2067 to (12.01, 5.78, 90) mm, rotated rx -180 ry 0 rz -180 deg; joints [-159.874, -54.235, -90.748, 24.107, 57.399, -13.555]
  Call Extruder(19804.47766)
  MoveL 2068 to (10.42, 8.31, 90) mm, rotated rx -180 ry 0 rz 180 deg; joints [-159.432, -54.197, -90.855, 24.597, 57.567, -13.794]
  Call Extruder(19809.14185)
  MoveL 2069 to (8.31, 10.42, 90) mm, rotated rx 180 ry 0 rz 180 deg; joints [-159.021, -54.122, -91.071, 25.033, 57.794, -13.977]
  Call Extruder(19813.80547)
  MoveL 2070 to (5.78, 12.01, 90) mm, rotated rx 180 ry 0 rz 180 deg; joints [-158.657, -54.013, -91.386, 25.394, 58.068, -14.095]
  Call Extruder(19818.46905)
  MoveL 2071 to (2.97, 12.99, 90) mm, rotated rx -180 ry 0 rz 180 deg; joints [-158.359, -53.877, -91.783, 25.664, 58.375, -14.142]
  Call Extruder(19823.13301)
  MoveL 2072 to (0, 13.33, 90) mm, rotated rx 180 ry 0 rz 180 deg; joints [-158.143, -53.719, -92.243, 25.83, 58.701, -14.116]
  Call Extruder(19827.79696)
  MoveL 2073 to (-2.97, 12.99, 90) mm, rotated rx 180 ry 0 rz 180 deg; joints [-158.019, -53.549, -92.744, 25.883, 59.029, -14.019]
  Call Extruder(19832.46052)
  MoveL 2074 to (-5.78, 12.01, 90) mm, rotated rx -180 ry 0 rz -180 deg; joints [-157.997, -53.375, -93.262, 25.818, 59.343, -13.858]
  Call Extruder(19837.12416)
  MoveL 2075 to (-8.31, 10.42, 90) mm, rotated rx -180 ry 0 rz 180 deg; joints [-158.08, -53.205, -93.77, 25.638, 59.629, -13.64]
  Call Extruder(19841.78835)
  MoveL 2076 to (-10.42, 8.31, 90) mm, rotated rx 180 ry 0 rz 180 deg; joints [-158.266, -53.049, -94.242, 25.349, 59.87, -13.377]
  Call Extruder(19846.45197)
  MoveL 2077 to (-12.01, 5.78, 90) mm, rotated rx -180 ry 0 rz 180 deg; joints [-158.549, -52.914, -94.655, 24.964, 60.057, -13.082]
  Call Extruder(19851.11554)
  MoveL 2078 to (-13, 2.97, 90) mm, rotated rx 180 ry 0 rz -180 deg; joints [-158.913, -52.806, -94.987, 24.5, 60.179, -12.769]
  Call Extruder(19855.77950)
  MoveL 2079 to (-13.33, 0, 90) mm, rotated rx -180 ry 0 rz 180 deg; joints [-159.341, -52.73, -95.22, 23.981, 60.229, -12.455]
  Call Extruder(19860.44345)
  MoveL 2080 to (-12.99, -2.97, 90) mm, rotated rx 180 ry 0 rz 180 deg; joints [-159.811, -52.691, -95.343, 23.434, 60.206, -12.154]
  Call Extruder(19865.10701)
  MoveL 2081 to (-12.01, -5.78, 90) mm, rotated rx 180 ry 0 rz -180 deg; joints [-160.294, -52.689, -95.349, 22.888, 60.108, -11.881]
  Call Extruder(19869.77065)
  MoveL 2082 to (-10.42, -8.31, 90) mm, rotated rx 180 ry 0 rz 180 deg; joints [-160.766, -52.725, -95.238, 22.371, 59.943, -11.648]
  Call Extruder(19874.43484)
  MoveL 2083 to (-8.31, -10.42, 90) mm, rotated rx 180 ry 0 rz -180 deg; joints [-161.2, -52.797, -95.015, 21.913, 59.716, -11.467]
  Call Extruder(19879.09847)
  MoveL 2084 to (-5.78, -12.01, 90) mm, rotated rx 180 ry 0 rz 180 deg; joints [-161.572, -52.902, -94.692, 21.538, 59.44, -11.347]
  Call Extruder(19883.76203)
  MoveL 2085 to (-2.97, -12.99, 90) mm, rotated rx 180 ry 0 rz 180 deg; joints [-161.863, -53.035, -94.286, 21.265, 59.129, -11.293]
  Call Extruder(19888.42599)
  MoveL 2086 to (0, -13.33, 90) mm, rotated rx -180 ry 0 rz -180 deg; joints [-162.059, -53.189, -93.818, 21.108, 58.799, -11.309]
  Call Extruder(19891.74156)
  MoveL 2087 to (2.11, -13.09, 90) mm, rotated rx -180 ry 0 rz -180 deg; joints [-162.125, -53.309, -93.459, 21.084, 58.562, -11.37]
  Set speed (130.0 mm/s)
  MoveL 2088 to (2.11, -13.09, 95) mm, rotated rx 180 ry 0 rz 180 deg; joints [-162.125, -52.545, -93.789, 21.181, 58.158, -11.554]
  MoveL 2089 to (-26.25, -4.54, 95) mm, rotated rx 180 ry 0 rz -180 deg; joints [-159.288, -51.206, -97.871, 23.786, 61.27, -11.962]
  Call Extruder(19893.97417)
  Set speed (60.0 mm/s)
  MoveL 2090 to (-26.09, -5.96, 95) mm, rotated rx 180 ry 0 rz 180 deg; joints [-159.522, -51.187, -97.929, 23.516, 61.259, -11.818]
  Call Extruder(19903.33897)
  MoveL 2091 to (-24.11, -11.61, 95) mm, rotated rx -180 ry 0 rz 180 deg; joints [-160.532, -51.184, -97.941, 22.385, 61.064, -11.27]
  Call Extruder(19912.70389)
  MoveL 2092 to (-20.93, -16.69, 95) mm, rotated rx 180 ry 0 rz 180 deg; joints [-161.513, -51.256, -97.712, 21.315, 60.731, -10.8]
  Call Extruder(19922.06909)
  MoveL 2093 to (-16.69, -20.93, 95) mm, rotated rx 180 ry 0 rz 180 deg; joints [-162.406, -51.401, -97.255, 20.369, 60.275, -10.431]
  Call Extruder(19931.43401)
  MoveL 2094 to (-11.61, -24.12, 95) mm, rotated rx 180 ry 0 rz 180 deg; joints [-163.159, -51.613, -96.596, 19.602, 59.72, -10.18]
  Call Extruder(19940.79880)
  MoveL 2095 to (-5.96, -26.09, 95) mm, rotated rx 180 ry 0 rz 180 deg; joints [-163.733, -51.882, -95.77, 19.054, 59.094, -10.06]
  Call Extruder(19950.16391)
  MoveL 2096 to (0, -26.77, 95) mm, rotated rx 180 ry 0 rz 180 deg; joints [-164.103, -52.197, -94.823, 18.753, 58.43, -10.079]
  Call Extruder(19956.48622)
  MoveL 2097 to (4.02, -26.31, 95) mm, rotated rx 180 ry 0 rz 180 deg; joints [-164.208, -52.428, -94.135, 18.722, 57.98, -10.187]
  Call Extruder(19959.52902)
  MoveL 2098 to (5.96, -26.09, 95) mm, rotated rx 180 ry 0 rz 180 deg; joints [-164.258, -52.541, -93.803, 18.708, 57.763, -10.24]
  Call Extruder(19968.89382)
  MoveL 2099 to (11.61, -24.11, 95) mm, rotated rx 180 ry 0 rz 180 deg; joints [-164.201, -52.898, -92.762, 18.916, 57.126, -10.537]
  Call Extruder(19978.25873)
  MoveL 2100 to (16.69, -20.93, 95) mm, rotated rx 180 ry 0 rz 180 deg; joints [-163.944, -53.25, -91.753, 19.358, 56.554, -10.959]
  Call Extruder(19987.62393)
  MoveL 2101 to (20.93, -16.69, 95) mm, rotated rx 180 ry 0 rz 180 deg; joints [-163.508, -53.579, -90.824, 20.007, 56.073, -11.487]
  Call Extruder(19996.98885)
  MoveL 2102 to (24.12, -11.61, 95) mm, rotated rx 180 ry 0 rz 180 deg; joints [-162.92, -53.867, -90.019, 20.824, 55.71, -12.095]
  Call Extruder(20006.35365)
  MoveL 2103 to (26.09, -5.96, 95) mm, rotated rx -180 ry 0 rz -180 deg; joints [-162.209, -54.099, -89.378, 21.767, 55.481, -12.75]
  Call Extruder(20015.71875)
  MoveL 2104 to (26.77, 0, 95) mm, rotated rx 180 ry 0 rz -180 deg; joints [-161.41, -54.263, -88.928, 22.787, 55.397, -13.418]
  Call Extruder(20025.08385)
  MoveL 2105 to (26.09, 5.96, 95) mm, rotated rx -180 ry 0 rz 180 deg; joints [-160.556, -54.349, -88.693, 23.835, 55.463, -14.061]
  Call Extruder(20034.44866)
  MoveL 2106 to (24.11, 11.61, 95) mm, rotated rx 180 ry 0 rz 180 deg; joints [-159.683, -54.353, -88.682, 24.862, 55.673, -14.645]
  Call Extruder(20043.81357)
  MoveL 2107 to (20.93, 16.69, 95) mm, rotated rx 180 ry 0 rz 180 deg; joints [-158.826, -54.275, -88.895, 25.824, 56.016, -15.137]
  Call Extruder(20053.17877)
  MoveL 2108 to (16.69, 20.93, 95) mm, rotated rx 180 ry 0 rz 180 deg; joints [-158.019, -54.119, -89.324, 26.679, 56.473, -15.511]
  Call Extruder(20062.54369)
  MoveL 2109 to (11.61, 24.11, 95) mm, rotated rx 180 ry 0 rz 180 deg; joints [-157.299, -53.893, -89.948, 27.39, 57.022, -15.75]
  Call Extruder(20071.90849)
  MoveL 2110 to (5.96, 26.09, 95) mm, rotated rx -180 ry 0 rz 180 deg; joints [-156.697, -53.61, -90.738, 27.927, 57.634, -15.842]
  Call Extruder(20081.27360)
  MoveL 2111 to (0, 26.77, 95) mm, rotated rx 180 ry 0 rz 180 deg; joints [-156.245, -53.284, -91.656, 28.266, 58.281, -15.785]
  Call Extruder(20090.63870)
  MoveL 2112 to (-5.96, 26.09, 95) mm, rotated rx 180 ry 0 rz 180 deg; joints [-155.969, -52.934, -92.66, 28.388, 58.93, -15.584]
  Call Extruder(20100.00349)
  MoveL 2113 to (-11.61, 24.11, 95) mm, rotated rx -180 ry 0 rz 180 deg; joints [-155.891, -52.576, -93.699, 28.283, 59.551, -15.252]
  Call Extruder(20109.36841)
  MoveL 2114 to (-16.69, 20.93, 95) mm, rotated rx 180 ry 0 rz -180 deg; joints [-156.025, -52.23, -94.724, 27.947, 60.114, -14.807]
  Call Extruder(20118.73362)
  MoveL 2115 to (-20.93, 16.69, 95) mm, rotated rx 180 ry 0 rz 180 deg; joints [-156.374, -51.912, -95.681, 27.39, 60.593, -14.274]
  Call Extruder(20128.09853)
  MoveL 2116 to (-24.11, 11.61, 95) mm, rotated rx -180 ry 0 rz 180 deg; joints [-156.928, -51.637, -96.521, 26.63, 60.963, -13.679]
  Call Extruder(20137.46333)
  MoveL 2117 to (-26.09, 5.96, 95) mm, rotated rx -180 ry 0 rz 180 deg; joints [-157.665, -51.419, -97.198, 25.699, 61.205, -13.051]
  Call Extruder(20146.82844)
  MoveL 2118 to (-26.77, 0, 95) mm, rotated rx 180 ry 0 rz -180 deg; joints [-158.546, -51.267, -97.677, 24.642, 61.306, -12.421]
  Call Extruder(20151.61718)
  MoveL 2119 to (-26.42, -3.05, 95) mm, rotated rx 180 ry 0 rz 180 deg; joints [-159.044, -51.226, -97.808, 24.068, 61.282, -12.113]
  Set speed (130.0 mm/s)
  MoveL 2120 to (-41.86, -6.3, 95) mm, rotated rx -180 ry 0 rz 180 deg; joints [-158.606, -50.433, -100.394, 24.166, 63.009, -11.511]
  Call Extruder(20156.61502)
  Set speed (60.0 mm/s)
  MoveL 2121 to (-41.5, -9.47, 95) mm, rotated rx 180 ry 0 rz 180 deg; joints [-159.151, -50.394, -100.528, 23.546, 62.987, -11.195]
  Call Extruder(20171.51067)
  MoveL 2122 to (-38.36, -18.47, 95) mm, rotated rx 180 ry 0 rz 180 deg; joints [-160.835, -50.388, -100.547, 21.683, 62.685, -10.34]
  Call Extruder(20186.40653)
  MoveL 2123 to (-33.28, -26.54, 95) mm, rotated rx 180 ry 0 rz 180 deg; joints [-162.466, -50.499, -100.174, 19.921, 62.157, -9.607]
  Call Extruder(20201.30234)
  MoveL 2124 to (-26.54, -33.28, 95) mm, rotated rx 180 ry 0 rz -180 deg; joints [-163.93, -50.723, -99.43, 18.373, 61.429, -9.025]
  Call Extruder(20216.19820)
  MoveL 2125 to (-18.47, -38.36, 95) mm, rotated rx -180 ry 0 rz 180 deg; joints [-165.137, -51.052, -98.36, 17.134, 60.539, -8.622]
  Call Extruder(20231.09384)
  MoveL 2126 to (-9.47, -41.5, 95) mm, rotated rx -180 ry 0 rz -180 deg; joints [-166.024, -51.474, -97.028, 16.272, 59.536, -8.418]
  Call Extruder(20245.98972)
  MoveL 2127 to (0, -42.57, 95) mm, rotated rx -180 ry 0 rz 180 deg; joints [-166.562, -51.969, -95.508, 15.822, 58.472, -8.429]
  Call Extruder(20255.07758)
  MoveL 2128 to (5.78, -41.92, 95) mm, rotated rx -180 ry 0 rz 180 deg; joints [-166.675, -52.299, -94.518, 15.802, 57.82, -8.571]
  Call Extruder(20260.88559)
  MoveL 2129 to (9.47, -41.51, 95) mm, rotated rx 180 ry 0 rz 180 deg; joints [-166.745, -52.514, -93.881, 15.792, 57.404, -8.663]
  Call Extruder(20275.78125)
  MoveL 2130 to (18.47, -38.36, 95) mm, rotated rx -180 ry 0 rz 180 deg; joints [-166.591, -53.084, -92.229, 16.168, 56.386, -9.118]
  Call Extruder(20290.67710)
  MoveL 2131 to (26.54, -33.28, 95) mm, rotated rx 180 ry 0 rz 180 deg; joints [-166.133, -53.647, -90.633, 16.913, 55.472, -9.779]
  Call Extruder(20305.57292)
  MoveL 2132 to (33.28, -26.54, 95) mm, rotated rx -180 ry 0 rz 180 deg; joints [-165.409, -54.176, -89.168, 17.977, 54.707, -10.618]
  Call Extruder(20320.46877)
  MoveL 2133 to (38.36, -18.47, 95) mm, rotated rx -180 ry 0 rz 180 deg; joints [-164.468, -54.64, -87.903, 19.296, 54.13, -11.594]
  Call Extruder(20335.36442)
  MoveL 2134 to (41.5, -9.47, 95) mm, rotated rx 180 ry 0 rz 180 deg; joints [-163.355, -55.015, -86.896, 20.8, 53.769, -12.654]
  Call Extruder(20350.26029)
  MoveL 2135 to (42.57, 0, 95) mm, rotated rx 180 ry 0 rz 180 deg; joints [-162.12, -55.28, -86.191, 22.411, 53.643, -13.738]
  Call Extruder(20365.15617)
  MoveL 2136 to (41.51, 9.47, 95) mm, rotated rx -180 ry 0 rz 180 deg; joints [-160.81, -55.42, -85.822, 24.052, 53.754, -14.783]
  Call Extruder(20380.05183)
  MoveL 2137 to (38.36, 18.47, 95) mm, rotated rx 180 ry 0 rz 180 deg; joints [-159.475, -55.426, -85.804, 25.65, 54.096, -15.727]
  Call Extruder(20394.94767)
  MoveL 2138 to (33.29, 26.54, 95) mm, rotated rx 180 ry 0 rz 180 deg; joints [-158.16, -55.3, -86.139, 27.137, 54.647, -16.518]
  Call Extruder(20409.84350)
  MoveL 2139 to (26.54, 33.28, 95) mm, rotated rx 180 ry 0 rz 180 deg; joints [-156.916, -55.047, -86.812, 28.454, 55.378, -17.113]
  Call Extruder(20424.73934)
  MoveL 2140 to (18.47, 38.36, 95) mm, rotated rx 180 ry 0 rz -180 deg; joints [-155.789, -54.682, -87.791, 29.552, 56.251, -17.484]
  Call Extruder(20439.63501)
  MoveL 2141 to (9.47, 41.5, 95) mm, rotated rx -180 ry 0 rz -180 deg; joints [-154.828, -54.225, -89.033, 30.391, 57.221, -17.616]
  Call Extruder(20454.53088)
  MoveL 2142 to (0, 42.57, 95) mm, rotated rx 180 ry 0 rz 180 deg; joints [-154.081, -53.702, -90.48, 30.935, 58.241, -17.508]
  Call Extruder(20469.42675)
  MoveL 2143 to (-9.47, 41.51, 95) mm, rotated rx -180 ry 0 rz 180 deg; joints [-153.594, -53.14, -92.067, 31.158, 59.264, -17.172]
  Call Extruder(20484.32240)
  MoveL 2144 to (-18.47, 38.36, 95) mm, rotated rx 180 ry 0 rz 180 deg; joints [-153.408, -52.57, -93.717, 31.039, 60.243, -16.63]
  Call Extruder(20499.21826)
  MoveL 2145 to (-26.54, 33.29, 95) mm, rotated rx 180 ry 0 rz 180 deg; joints [-153.557, -52.021, -95.35, 30.563, 61.133, -15.913]
  Call Extruder(20514.11407)
  MoveL 2146 to (-33.29, 26.54, 95) mm, rotated rx 180 ry 0 rz 180 deg; joints [-154.059, -51.52, -96.885, 29.731, 61.892, -15.06]
  Call Extruder(20529.00992)
  MoveL 2147 to (-38.36, 18.47, 95) mm, rotated rx -180 ry 0 rz 180 deg; joints [-154.913, -51.09, -98.239, 28.559, 62.485, -14.115]
  Call Extruder(20543.90558)
  MoveL 2148 to (-41.5, 9.47, 95) mm, rotated rx -180 ry 0 rz 180 deg; joints [-156.091, -50.751, -99.337, 27.088, 62.879, -13.125]
  Call Extruder(20558.80146)
  MoveL 2149 to (-42.57, 0, 95) mm, rotated rx 180 ry 0 rz -180 deg; joints [-157.533, -50.516, -100.116, 25.386, 63.051, -12.137]
  Call Extruder(20566.35574)
  MoveL 2150 to (-42.03, -4.8, 95) mm, rotated rx 180 ry 0 rz 180 deg; joints [-158.35, -50.452, -100.33, 24.456, 63.019, -11.659]
  Set speed (130.0 mm/s)
  MoveL 2151 to (-54.1, -7.67, 95) mm, rotated rx 180 ry 0 rz 180 deg; joints [-158.024, -49.872, -102.333, 24.521, 64.379, -11.159]
  Call Extruder(20570.42837)
  Set speed (30.0 mm/s)
  MoveL 2152 to (-53.59, -12.23, 95) mm, rotated rx 180 ry 0 rz 180 deg; joints [-158.835, -49.818, -102.527, 23.61, 64.352, -10.713]
  Call Extruder(20581.35850)
  MoveL 2153 to (-49.53, -23.85, 95) mm, rotated rx -180 ry 0 rz 180 deg; joints [-161.095, -49.811, -102.553, 21.135, 63.97, -9.628]
  Call Extruder(20592.28879)
  MoveL 2154 to (-42.98, -34.27, 95) mm, rotated rx 180 ry 0 rz 180 deg; joints [-163.275, -49.949, -102.06, 18.793, 63.29, -8.696]
  Call Extruder(20603.21890)
  MoveL 2155 to (-34.27, -42.98, 95) mm, rotated rx 180 ry 0 rz 180 deg; joints [-165.21, -50.231, -101.08, 16.75, 62.345, -7.952]
  Call Extruder(20614.14919)
  MoveL 2156 to (-23.85, -49.53, 95) mm, rotated rx -180 ry 0 rz 180 deg; joints [-166.774, -50.648, -99.678, 15.137, 61.188, -7.428]
  Call Extruder(20625.07932)
  MoveL 2157 to (-12.23, -53.59, 95) mm, rotated rx -180 ry 0 rz 180 deg; joints [-167.889, -51.184, -97.939, 14.037, 59.883, -7.151]
  Call Extruder(20636.00954)
  MoveL 2158 to (0, -54.97, 95) mm, rotated rx 180 ry 0 rz 180 deg; joints [-168.526, -51.819, -95.964, 13.491, 58.502, -7.145]
  Call Extruder(20642.40671)
  MoveL 2159 to (7.16, -54.16, 95) mm, rotated rx 180 ry 0 rz 180 deg; joints [-168.628, -52.225, -94.737, 13.492, 57.691, -7.308]
  Call Extruder(20646.93976)
  MoveL 2160 to (12.23, -53.59, 95) mm, rotated rx 180 ry 0 rz 180 deg; joints [-168.697, -52.522, -93.859, 13.497, 57.117, -7.425]
  Call Extruder(20657.86990)
  MoveL 2161 to (23.85, -49.53, 95) mm, rotated rx 180 ry 0 rz 180 deg; joints [-168.436, -53.258, -91.73, 14.026, 55.799, -7.993]
  Call Extruder(20668.80018)
  MoveL 2162 to (34.27, -42.98, 95) mm, rotated rx 180 ry 0 rz 180 deg; joints [-167.797, -53.99, -89.679, 15.027, 54.616, -8.836]
  Call Extruder(20679.73030)
  MoveL 2163 to (42.98, -34.27, 95) mm, rotated rx 180 ry 0 rz 180 deg; joints [-166.837, -54.678, -87.801, 16.429, 53.626, -9.919]
  Call Extruder(20690.66059)
  MoveL 2164 to (49.52, -23.85, 95) mm, rotated rx 180 ry 0 rz 180 deg; joints [-165.618, -55.284, -86.182, 18.149, 52.881, -11.19]
  Call Extruder(20701.59072)
  MoveL 2165 to (53.59, -12.23, 95) mm, rotated rx -180 ry 0 rz -180 deg; joints [-164.2, -55.774, -84.892, 20.095, 52.418, -12.578]
  Call Extruder(20712.52094)
  MoveL 2166 to (54.97, 0, 95) mm, rotated rx 180 ry 0 rz 180 deg; joints [-162.641, -56.12, -83.991, 22.167, 52.259, -14.002]
  Call Extruder(20723.45116)
  MoveL 2167 to (53.59, 12.23, 95) mm, rotated rx 180 ry 0 rz 180 deg; joints [-160.996, -56.303, -83.519, 24.264, 52.41, -15.374]
  Call Extruder(20734.38131)
  MoveL 2168 to (49.52, 23.85, 95) mm, rotated rx 180 ry 0 rz -180 deg; joints [-159.322, -56.312, -83.496, 26.293, 52.859, -16.611]
  Call Extruder(20745.31158)
  MoveL 2169 to (42.98, 34.27, 95) mm, rotated rx 180 ry 0 rz 180 deg; joints [-157.673, -56.146, -83.925, 28.172, 53.578, -17.639]
  Call Extruder(20756.24171)
  MoveL 2170 to (34.27, 42.98, 95) mm, rotated rx -180 ry 0 rz 180 deg; joints [-156.102, -55.815, -84.785, 29.83, 54.527, -18.405]
  Call Extruder(20767.17198)
  MoveL 2171 to (23.85, 49.53, 95) mm, rotated rx 180 ry 0 rz 180 deg; joints [-154.667, -55.338, -86.038, 31.213, 55.654, -18.874]
  Call Extruder(20778.10213)
  MoveL 2172 to (12.23, 53.59, 95) mm, rotated rx -180 ry 0 rz 180 deg; joints [-153.426, -54.742, -87.628, 32.276, 56.903, -19.028]
  Call Extruder(20789.03235)
  MoveL 2173 to (0, 54.97, 95) mm, rotated rx 180 ry 0 rz 180 deg; joints [-152.438, -54.061, -89.484, 32.981, 58.213, -18.872]
  Call Extruder(20799.96257)
  MoveL 2174 to (-12.23, 53.59, 95) mm, rotated rx 180 ry 0 rz 180 deg; joints [-151.764, -53.332, -91.522, 33.295, 59.525, -18.422]
  Call Extruder(20810.89270)
  MoveL 2175 to (-23.85, 49.52, 95) mm, rotated rx 180 ry 0 rz 180 deg; joints [-151.463, -52.594, -93.648, 33.187, 60.779, -17.709]
  Call Extruder(20821.82299)
  MoveL 2176 to (-34.27, 42.98, 95) mm, rotated rx 180 ry 0 rz 180 deg; joints [-151.589, -51.886, -95.76, 32.634, 61.92, -16.774]
  Call Extruder(20832.75311)
  MoveL 2177 to (-42.98, 34.27, 95) mm, rotated rx 180 ry 0 rz -180 deg; joints [-152.179, -51.243, -97.752, 31.619, 62.899, -15.667]
  Call Extruder(20843.68339)
  MoveL 2178 to (-49.53, 23.85, 95) mm, rotated rx -180 ry 0 rz -180 deg; joints [-153.248, -50.696, -99.519, 30.149, 63.668, -14.448]
  Call Extruder(20854.61353)
  MoveL 2179 to (-53.59, 12.23, 95) mm, rotated rx 180 ry 0 rz 180 deg; joints [-154.769, -50.267, -100.958, 28.263, 64.186, -13.175]
  Call Extruder(20865.54375)
  MoveL 2180 to (-54.97, 0, 95) mm, rotated rx -180 ry 0 rz -180 deg; joints [-156.673, -49.971, -101.983, 26.041, 64.422, -11.912]
  Call Extruder(20871.06937)
  MoveL 2181 to (-54.27, -6.18, 95) mm, rotated rx 180 ry 0 rz 180 deg; joints [-157.76, -49.891, -102.268, 24.818, 64.387, -11.305]
  Set speed (130.0 mm/s)
  MoveL 2182 to (-49.9, -9.51, 95) mm, rotated rx 180 ry 0 rz 180 deg; joints [-158.616, -50.021, -101.809, 23.95, 63.922, -11.048]
  MoveL 2183 to (2.53, -13.05, 95) mm, rotated rx 180 ry 0 rz 180 deg; joints [-162.139, -52.57, -93.718, 21.176, 58.111, -11.566]
  Call Extruder(20871.76173)
  Set speed (80.0 mm/s)
  MoveL 2184 to (2.97, -12.99, 95) mm, rotated rx 180 ry 0 rz -180 deg; joints [-162.152, -52.595, -93.643, 21.171, 58.062, -11.579]
  Call Extruder(20876.42529)
  MoveL 2185 to (5.78, -12.01, 95) mm, rotated rx 180 ry 0 rz 180 deg; joints [-162.141, -52.773, -93.124, 21.262, 57.747, -11.731]
  Call Extruder(20881.08891)
  MoveL 2186 to (8.31, -10.42, 95) mm, rotated rx -180 ry 0 rz -180 deg; joints [-162.027, -52.948, -92.619, 21.47, 57.463, -11.945]
  Call Extruder(20885.75311)
  MoveL 2187 to (10.42, -8.31, 95) mm, rotated rx -180 ry 0 rz 180 deg; joints [-161.819, -53.11, -92.153, 21.784, 57.224, -12.208]
  Call Extruder(20890.41674)
  MoveL 2188 to (12.01, -5.78, 95) mm, rotated rx -180 ry 0 rz 180 deg; joints [-161.529, -53.252, -91.748, 22.185, 57.042, -12.508]
  Call Extruder(20895.08030)
  MoveL 2189 to (13, -2.97, 95) mm, rotated rx 180 ry 0 rz -180 deg; joints [-161.171, -53.366, -91.425, 22.653, 56.927, -12.83]
  Call Extruder(20899.74426)
  MoveL 2190 to (13.33, 0, 95) mm, rotated rx 180 ry 0 rz 180 deg; joints [-160.763, -53.446, -91.198, 23.165, 56.884, -13.158]
  Call Extruder(20904.40821)
  MoveL 2191 to (13, 2.97, 95) mm, rotated rx 180 ry 0 rz 180 deg; joints [-160.324, -53.488, -91.079, 23.695, 56.914, -13.473]
  Call Extruder(20909.07178)
  MoveL 2192 to (12.01, 5.78, 95) mm, rotated rx -180 ry 0 rz -180 deg; joints [-159.874, -53.49, -91.073, 24.218, 57.017, -13.759]
  Call Extruder(20913.73541)
  MoveL 2193 to (10.42, 8.31, 95) mm, rotated rx 180 ry 0 rz 180 deg; joints [-159.432, -53.452, -91.181, 24.709, 57.186, -14.002]
  Call Extruder(20918.39960)
  MoveL 2194 to (8.31, 10.42, 95) mm, rotated rx 180 ry 0 rz 180 deg; joints [-159.021, -53.375, -91.398, 25.146, 57.413, -14.188]
  Call Extruder(20923.06322)
  MoveL 2195 to (5.78, 12.01, 95) mm, rotated rx 180 ry 0 rz 180 deg; joints [-158.657, -53.264, -91.712, 25.508, 57.687, -14.309]
  Call Extruder(20927.72680)
  MoveL 2196 to (2.97, 13, 95) mm, rotated rx -180 ry 0 rz 180 deg; joints [-158.359, -53.125, -92.11, 25.779, 57.993, -14.358]
  Call Extruder(20932.39075)
  MoveL 2197 to (0, 13.33, 95) mm, rotated rx 180 ry 0 rz 180 deg; joints [-158.143, -52.964, -92.571, 25.944, 58.317, -14.334]
  Call Extruder(20937.05470)
  MoveL 2198 to (-2.97, 12.99, 95) mm, rotated rx -180 ry 0 rz 180 deg; joints [-158.019, -52.791, -93.073, 25.997, 58.643, -14.239]
  Call Extruder(20941.71827)
  MoveL 2199 to (-5.78, 12.01, 95) mm, rotated rx 180 ry 0 rz -180 deg; joints [-157.997, -52.613, -93.591, 25.931, 58.954, -14.078]
  Call Extruder(20946.38190)
  MoveL 2200 to (-8.31, 10.42, 95) mm, rotated rx 180 ry 0 rz 180 deg; joints [-158.08, -52.44, -94.1, 25.75, 59.236, -13.859]
  Call Extruder(20951.04610)
  MoveL 2201 to (-10.42, 8.31, 95) mm, rotated rx 180 ry 0 rz 180 deg; joints [-158.266, -52.28, -94.573, 25.459, 59.475, -13.594]
  Call Extruder(20955.70971)
  MoveL 2202 to (-12.01, 5.78, 95) mm, rotated rx -180 ry 0 rz -180 deg; joints [-158.549, -52.142, -94.987, 25.072, 59.658, -13.297]
  Call Extruder(20960.37329)
  MoveL 2203 to (-13, 2.97, 95) mm, rotated rx -180 ry 0 rz -180 deg; joints [-158.913, -52.031, -95.319, 24.606, 59.777, -12.982]
  Call Extruder(20965.03724)
  MoveL 2204 to (-13.33, 0, 95) mm, rotated rx 180 ry 0 rz -180 deg; joints [-159.341, -51.954, -95.553, 24.086, 59.824, -12.664]
  Call Extruder(20969.70119)
  MoveL 2205 to (-12.99, -2.97, 95) mm, rotated rx -180 ry 0 rz 180 deg; joints [-159.811, -51.913, -95.677, 23.536, 59.798, -12.359]
  Call Extruder(20974.36476)
  MoveL 2206 to (-12.01, -5.78, 95) mm, rotated rx 180 ry 0 rz 180 deg; joints [-160.294, -51.911, -95.682, 22.988, 59.699, -12.081]
  Call Extruder(20979.02839)
  MoveL 2207 to (-10.42, -8.31, 95) mm, rotated rx 180 ry 0 rz 180 deg; joints [-160.766, -51.948, -95.571, 22.47, 59.533, -11.844]
  Call Extruder(20983.69259)
  MoveL 2208 to (-8.31, -10.42, 95) mm, rotated rx -180 ry 0 rz 180 deg; joints [-161.2, -52.022, -95.347, 22.01, 59.306, -11.659]
  Call Extruder(20988.35621)
  MoveL 2209 to (-5.78, -12.01, 95) mm, rotated rx 180 ry 0 rz 180 deg; joints [-161.572, -52.13, -95.024, 21.634, 59.031, -11.535]
  Call Extruder(20993.01978)
  MoveL 2210 to (-2.97, -13, 95) mm, rotated rx 180 ry 0 rz 180 deg; joints [-161.863, -52.265, -94.617, 21.361, 58.721, -11.479]
  Call Extruder(20997.68372)
  MoveL 2211 to (0, -13.33, 95) mm, rotated rx 180 ry 0 rz -180 deg; joints [-162.059, -52.423, -94.149, 21.204, 58.393, -11.493]
  Call Extruder(21001.65534)
  MoveL 2212 to (2.53, -13.05, 95) mm, rotated rx 180 ry 0 rz 180 deg; joints [-162.139, -52.57, -93.718, 21.176, 58.111, -11.566]
  Set speed (130.0 mm/s)
  MoveL 2213 to (2.53, -13.04, 100) mm, rotated rx 180 ry 0 rz 180 deg; joints [-162.139, -51.808, -94.038, 21.276, 57.7, -11.754]
  MoveL 2214 to (-26.25, -4.54, 100) mm, rotated rx 180 ry 0 rz 180 deg; joints [-159.288, -50.411, -98.199, 23.89, 60.844, -12.177]
  Call Extruder(21003.88795)
  Set speed (60.0 mm/s)
  MoveL 2215 to (-26.09, -5.96, 100) mm, rotated rx -180 ry 0 rz 180 deg; joints [-159.522, -50.393, -98.258, 23.62, 60.831, -12.031]
  Call Extruder(21013.25274)
  MoveL 2216 to (-24.11, -11.61, 100) mm, rotated rx -180 ry 0 rz 180 deg; joints [-160.532, -50.389, -98.27, 22.484, 60.633, -11.474]
  Call Extruder(21022.61766)
  MoveL 2217 to (-20.93, -16.69, 100) mm, rotated rx 180 ry 0 rz 180 deg; joints [-161.513, -50.463, -98.04, 21.411, 60.298, -10.995]
  Call Extruder(21031.98287)
  MoveL 2218 to (-16.69, -20.93, 100) mm, rotated rx -180 ry 0 rz 180 deg; joints [-162.406, -50.612, -97.582, 20.462, 59.842, -10.617]
  Call Extruder(21041.34778)
  MoveL 2219 to (-11.61, -24.12, 100) mm, rotated rx -180 ry 0 rz 180 deg; joints [-163.159, -50.829, -96.922, 19.692, 59.288, -10.359]
  Call Extruder(21050.71258)
  MoveL 2220 to (-5.96, -26.09, 100) mm, rotated rx -180 ry 0 rz 180 deg; joints [-163.733, -51.105, -96.094, 19.144, 58.666, -10.233]
  Call Extruder(21060.07769)
  MoveL 2221 to (0, -26.77, 100) mm, rotated rx 180 ry 0 rz 180 deg; joints [-164.103, -51.427, -95.145, 18.842, 58.006, -10.249]
  Call Extruder(21067.05603)
  MoveL 2222 to (4.44, -26.27, 100) mm, rotated rx 180 ry 0 rz 180 deg; joints [-164.219, -51.688, -94.384, 18.809, 57.513, -10.367]
  Call Extruder(21069.44278)
  MoveL 2223 to (5.96, -26.09, 100) mm, rotated rx 180 ry 0 rz 180 deg; joints [-164.258, -51.779, -94.123, 18.799, 57.344, -10.408]
  Call Extruder(21078.80759)
  MoveL 2224 to (11.61, -24.12, 100) mm, rotated rx 180 ry 0 rz 180 deg; joints [-164.201, -52.143, -93.081, 19.008, 56.714, -10.706]
  Call Extruder(21088.17250)
  MoveL 2225 to (16.69, -20.93, 100) mm, rotated rx 180 ry 0 rz 180 deg; joints [-163.944, -52.502, -92.07, 19.453, 56.148, -11.131]
  Call Extruder(21097.53771)
  MoveL 2226 to (20.93, -16.69, 100) mm, rotated rx 180 ry 0 rz 180 deg; joints [-163.508, -52.838, -91.14, 20.106, 55.674, -11.663]
  Call Extruder(21106.90263)
  MoveL 2227 to (24.11, -11.61, 100) mm, rotated rx -180 ry 0 rz 180 deg; joints [-162.92, -53.131, -90.335, 20.927, 55.316, -12.277]
  Call Extruder(21116.26742)
  MoveL 2228 to (26.09, -5.96, 100) mm, rotated rx 180 ry 0 rz -180 deg; joints [-162.209, -53.367, -89.692, 21.874, 55.093, -12.939]
  Call Extruder(21125.63252)
  MoveL 2229 to (26.77, 0, 100) mm, rotated rx -180 ry 0 rz -180 deg; joints [-161.41, -53.534, -89.242, 22.899, 55.015, -13.614]
  Call Extruder(21134.99763)
  MoveL 2230 to (26.09, 5.96, 100) mm, rotated rx 180 ry 0 rz 180 deg; joints [-160.556, -53.622, -89.007, 23.951, 55.084, -14.265]
  Call Extruder(21144.36243)
  MoveL 2231 to (24.12, 11.61, 100) mm, rotated rx 180 ry 0 rz 180 deg; joints [-159.683, -53.626, -88.995, 24.982, 55.297, -14.856]
  Call Extruder(21153.72734)
  MoveL 2232 to (20.93, 16.69, 100) mm, rotated rx 180 ry 0 rz 180 deg; joints [-158.826, -53.546, -89.209, 25.947, 55.642, -15.356]
  Call Extruder(21163.09255)
  MoveL 2233 to (16.69, 20.93, 100) mm, rotated rx 180 ry 0 rz 180 deg; joints [-158.019, -53.387, -89.638, 26.804, 56.1, -15.737]
  Call Extruder(21172.45746)
  MoveL 2234 to (11.61, 24.11, 100) mm, rotated rx 180 ry 0 rz 180 deg; joints [-157.299, -53.157, -90.263, 27.517, 56.649, -15.982]
  Call Extruder(21181.82227)
  MoveL 2235 to (5.96, 26.09, 100) mm, rotated rx 180 ry 0 rz 180 deg; joints [-156.697, -52.869, -91.054, 28.055, 57.259, -16.079]
  Call Extruder(21191.18737)
  MoveL 2236 to (0, 26.77, 100) mm, rotated rx 180 ry 0 rz 180 deg; joints [-156.245, -52.537, -91.974, 28.393, 57.902, -16.025]
  Call Extruder(21200.55247)
  MoveL 2237 to (-5.96, 26.09, 100) mm, rotated rx 180 ry 0 rz 180 deg; joints [-155.969, -52.179, -92.979, 28.514, 58.547, -15.827]
  Call Extruder(21209.91727)
  MoveL 2238 to (-11.61, 24.12, 100) mm, rotated rx 180 ry 0 rz 180 deg; joints [-155.891, -51.814, -94.02, 28.407, 59.163, -15.495]
  Call Extruder(21219.28219)
  MoveL 2239 to (-16.69, 20.93, 100) mm, rotated rx -180 ry 0 rz -180 deg; joints [-156.025, -51.46, -95.046, 28.069, 59.72, -15.05]
  Call Extruder(21228.64740)
  MoveL 2240 to (-20.93, 16.69, 100) mm, rotated rx 180 ry 0 rz 180 deg; joints [-156.374, -51.135, -96.005, 27.509, 60.191, -14.514]
  Call Extruder(21238.01231)
  MoveL 2241 to (-24.12, 11.61, 100) mm, rotated rx -180 ry 0 rz 180 deg; joints [-156.928, -50.854, -96.846, 26.745, 60.554, -13.914]
  Call Extruder(21247.37711)
  MoveL 2242 to (-26.09, 5.96, 100) mm, rotated rx 180 ry 0 rz 180 deg; joints [-157.665, -50.63, -97.525, 25.81, 60.789, -13.281]
  Call Extruder(21256.74221)
  MoveL 2243 to (-26.77, 0, 100) mm, rotated rx 180 ry 0 rz 180 deg; joints [-158.546, -50.474, -98.005, 24.75, 60.884, -12.643]
  Call Extruder(21261.53095)
  MoveL 2244 to (-26.42, -3.05, 100) mm, rotated rx 180 ry 0 rz 180 deg; joints [-159.044, -50.432, -98.136, 24.173, 60.857, -12.33]
  Set speed (130.0 mm/s)
  MoveL 2245 to (-41.86, -6.3, 100) mm, rotated rx 180 ry 0 rz 180 deg; joints [-158.606, -49.617, -100.729, 24.267, 62.569, -11.733]
  Call Extruder(21266.52880)
  Set speed (60.0 mm/s)
  MoveL 2246 to (-41.5, -9.47, 100) mm, rotated rx 180 ry 0 rz 180 deg; joints [-159.151, -49.576, -100.862, 23.645, 62.544, -11.413]
  Call Extruder(21281.42445)
  MoveL 2247 to (-38.36, -18.47, 100) mm, rotated rx 180 ry 0 rz 180 deg; joints [-160.835, -49.57, -100.882, 21.777, 62.236, -10.542]
  Call Extruder(21296.32030)
  MoveL 2248 to (-33.29, -26.54, 100) mm, rotated rx 180 ry 0 rz 180 deg; joints [-162.466, -49.684, -100.507, 20.008, 61.705, -9.793]
  Call Extruder(21311.21612)
  MoveL 2249 to (-26.54, -33.28, 100) mm, rotated rx -180 ry 0 rz -180 deg; joints [-163.93, -49.915, -99.761, 18.455, 60.978, -9.197]
  Call Extruder(21326.11197)
  MoveL 2250 to (-18.47, -38.36, 100) mm, rotated rx 180 ry 0 rz 180 deg; joints [-165.137, -50.254, -98.69, 17.213, 60.091, -8.781]
  Call Extruder(21341.00762)
  MoveL 2251 to (-9.47, -41.5, 100) mm, rotated rx 180 ry 0 rz 180 deg; joints [-166.024, -50.686, -97.355, 16.348, 59.093, -8.568]
  Call Extruder(21355.90350)
  MoveL 2252 to (0, -42.57, 100) mm, rotated rx 180 ry 0 rz 180 deg; joints [-166.562, -51.193, -95.832, 15.898, 58.037, -8.574]
  Call Extruder(21365.64740)
  MoveL 2253 to (6.2, -41.88, 100) mm, rotated rx 180 ry 0 rz 180 deg; joints [-166.683, -51.556, -94.768, 15.878, 57.344, -8.726]
  Call Extruder(21370.79936)
  MoveL 2254 to (9.47, -41.5, 100) mm, rotated rx 180 ry 0 rz 180 deg; joints [-166.745, -51.751, -94.202, 15.87, 56.978, -8.807]
  Call Extruder(21385.69503)
  MoveL 2255 to (18.47, -38.36, 100) mm, rotated rx -180 ry 0 rz 180 deg; joints [-166.591, -52.332, -92.547, 16.249, 55.971, -9.264]
  Call Extruder(21400.59088)
  MoveL 2256 to (26.54, -33.28, 100) mm, rotated rx 180 ry 0 rz 180 deg; joints [-166.133, -52.907, -90.949, 16.999, 55.066, -9.93]
  Call Extruder(21415.48669)
  MoveL 2257 to (33.29, -26.54, 100) mm, rotated rx 180 ry 0 rz 180 deg; joints [-165.409, -53.445, -89.482, 18.069, 54.311, -10.776]
  Call Extruder(21430.38255)
  MoveL 2258 to (38.36, -18.47, 100) mm, rotated rx -180 ry 0 rz 180 deg; joints [-164.468, -53.917, -88.216, 19.395, 53.743, -11.762]
  Call Extruder(21445.27820)
  MoveL 2259 to (41.5, -9.47, 100) mm, rotated rx -180 ry 0 rz 180 deg; joints [-163.355, -54.298, -87.208, 20.906, 53.391, -12.833]
  Call Extruder(21460.17407)
  MoveL 2260 to (42.57, 0, 100) mm, rotated rx -180 ry 0 rz 180 deg; joints [-162.12, -54.567, -86.502, 22.524, 53.271, -13.929]
  Call Extruder(21475.06994)
  MoveL 2261 to (41.51, 9.47, 100) mm, rotated rx -180 ry 0 rz -180 deg; joints [-160.81, -54.709, -86.133, 24.172, 53.389, -14.986]
  Call Extruder(21489.96561)
  MoveL 2262 to (38.36, 18.47, 100) mm, rotated rx -180 ry 0 rz 180 deg; joints [-159.475, -54.716, -86.115, 25.776, 53.735, -15.942]
  Call Extruder(21504.86145)
  MoveL 2263 to (33.29, 26.54, 100) mm, rotated rx 180 ry 0 rz 180 deg; joints [-158.16, -54.587, -86.45, 27.268, 54.29, -16.744]
  Call Extruder(21519.75728)
  MoveL 2264 to (26.54, 33.29, 100) mm, rotated rx 180 ry 0 rz 180 deg; joints [-156.916, -54.33, -87.123, 28.588, 55.023, -17.349]
  Call Extruder(21534.65312)
  MoveL 2265 to (18.47, 38.36, 100) mm, rotated rx 180 ry 0 rz -180 deg; joints [-155.789, -53.96, -88.104, 29.689, 55.895, -17.728]
  Call Extruder(21549.54878)
  MoveL 2266 to (9.47, 41.51, 100) mm, rotated rx 180 ry 0 rz 180 deg; joints [-154.828, -53.495, -89.347, 30.527, 56.862, -17.867]
  Call Extruder(21564.44465)
  MoveL 2267 to (0, 42.57, 100) mm, rotated rx 180 ry 0 rz 180 deg; joints [-154.081, -52.963, -90.796, 31.071, 57.878, -17.765]
  Call Extruder(21579.34053)
  MoveL 2268 to (-9.47, 41.51, 100) mm, rotated rx 180 ry 0 rz -180 deg; joints [-153.594, -52.39, -92.385, 31.293, 58.895, -17.433]
  Call Extruder(21594.23618)
  MoveL 2269 to (-18.47, 38.36, 100) mm, rotated rx -180 ry 0 rz 180 deg; joints [-153.408, -51.808, -94.037, 31.17, 59.865, -16.893]
  Call Extruder(21609.13203)
  MoveL 2270 to (-26.54, 33.29, 100) mm, rotated rx 180 ry 0 rz -180 deg; joints [-153.557, -51.247, -95.674, 30.691, 60.745, -16.175]
  Call Extruder(21624.02785)
  MoveL 2271 to (-33.28, 26.54, 100) mm, rotated rx 180 ry 0 rz -180 deg; joints [-154.059, -50.734, -97.211, 29.854, 61.493, -15.319]
  Call Extruder(21638.92370)
  MoveL 2272 to (-38.36, 18.47, 100) mm, rotated rx 180 ry 0 rz 180 deg; joints [-154.913, -50.293, -98.568, 28.677, 62.074, -14.368]
  Call Extruder(21653.81936)
  MoveL 2273 to (-41.5, 9.47, 100) mm, rotated rx -180 ry 0 rz 180 deg; joints [-156.091, -49.944, -99.669, 27.2, 62.456, -13.369]
  Call Extruder(21668.71523)
  MoveL 2274 to (-42.57, 0, 100) mm, rotated rx 180 ry 0 rz -180 deg; joints [-157.533, -49.702, -100.449, 25.491, 62.617, -12.369]
  Call Extruder(21676.26951)
  MoveL 2275 to (-42.03, -4.8, 100) mm, rotated rx -180 ry 0 rz 180 deg; joints [-158.35, -49.636, -100.664, 24.558, 62.581, -11.883]
  Set speed (130.0 mm/s)
  MoveL 2276 to (-54.1, -7.67, 100) mm, rotated rx -180 ry 0 rz -180 deg; joints [-158.024, -49.037, -102.673, 24.621, 63.928, -11.388]
  Call Extruder(21680.34214)
  Set speed (30.0 mm/s)
  MoveL 2277 to (-53.59, -12.23, 100) mm, rotated rx -180 ry 0 rz 180 deg; joints [-158.835, -48.981, -102.867, 23.707, 63.897, -10.935]
  Call Extruder(21691.27228)
  MoveL 2278 to (-49.52, -23.85, 100) mm, rotated rx -180 ry 0 rz 180 deg; joints [-161.095, -48.974, -102.893, 21.224, 63.507, -9.828]
  Call Extruder(21702.20256)
  MoveL 2279 to (-42.98, -34.27, 100) mm, rotated rx 180 ry 0 rz 180 deg; joints [-163.275, -49.117, -102.398, 18.874, 62.823, -8.875]
  Call Extruder(21713.13268)
  MoveL 2280 to (-34.27, -42.98, 100) mm, rotated rx 180 ry 0 rz 180 deg; joints [-165.21, -49.408, -101.416, 16.825, 61.879, -8.111]
  Call Extruder(21724.06296)
  MoveL 2281 to (-23.85, -49.52, 100) mm, rotated rx 180 ry 0 rz 180 deg; joints [-166.774, -49.838, -100.01, 15.206, 60.727, -7.571]
  Call Extruder(21734.99309)
  MoveL 2282 to (-12.23, -53.59, 100) mm, rotated rx 180 ry 0 rz 180 deg; joints [-167.889, -50.389, -98.268, 14.104, 59.431, -7.282]
  Call Extruder(21745.92332)
  MoveL 2283 to (0, -54.97, 100) mm, rotated rx 180 ry 0 rz 180 deg; joints [-168.526, -51.04, -96.289, 13.557, 58.06, -7.27]
  Call Extruder(21752.69332)
  MoveL 2284 to (7.58, -54.11, 100) mm, rotated rx 180 ry 0 rz -180 deg; joints [-168.633, -51.481, -94.987, 13.559, 57.209, -7.441]
  Call Extruder(21756.85354)
  MoveL 2285 to (12.23, -53.59, 100) mm, rotated rx 180 ry 0 rz 180 deg; joints [-168.697, -51.759, -94.18, 13.565, 56.687, -7.548]
  Call Extruder(21767.78368)
  MoveL 2286 to (23.85, -49.53, 100) mm, rotated rx -180 ry 0 rz 180 deg; joints [-168.436, -52.511, -92.048, 14.098, 55.382, -8.12]
  Call Extruder(21778.71396)
  MoveL 2287 to (34.27, -42.98, 100) mm, rotated rx -180 ry 0 rz 180 deg; joints [-167.797, -53.256, -89.994, 15.104, 54.211, -8.97]
  Call Extruder(21789.64408)
  MoveL 2288 to (42.98, -34.27, 100) mm, rotated rx -180 ry 0 rz 180 deg; joints [-166.837, -53.956, -88.114, 16.515, 53.234, -10.063]
  Call Extruder(21800.57436)
  MoveL 2289 to (49.53, -23.85, 100) mm, rotated rx 180 ry 0 rz 180 deg; joints [-165.618, -54.571, -86.493, 18.245, 52.5, -11.347]
  Call Extruder(21811.50450)
  MoveL 2290 to (53.59, -12.23, 100) mm, rotated rx -180 ry 0 rz -180 deg; joints [-164.2, -55.068, -85.202, 20.2, 52.047, -12.75]
  Call Extruder(21822.43472)
  MoveL 2291 to (54.97, 0, 100) mm, rotated rx 180 ry 0 rz 180 deg; joints [-162.641, -55.42, -84.301, 22.282, 51.897, -14.19]
  Call Extruder(21833.36494)
  MoveL 2292 to (53.59, 12.23, 100) mm, rotated rx 180 ry 0 rz 180 deg; joints [-160.996, -55.605, -83.828, 24.388, 52.056, -15.577]
  Call Extruder(21844.29508)
  MoveL 2293 to (49.52, 23.85, 100) mm, rotated rx -180 ry 0 rz -180 deg; joints [-159.322, -55.614, -83.805, 26.425, 52.511, -16.828]
  Call Extruder(21855.22536)
  MoveL 2294 to (42.98, 34.27, 100) mm, rotated rx 180 ry 0 rz 180 deg; joints [-157.673, -55.446, -84.234, 28.309, 53.234, -17.87]
  Call Extruder(21866.15548)
  MoveL 2295 to (34.27, 42.98, 100) mm, rotated rx 180 ry 0 rz 180 deg; joints [-156.102, -55.11, -85.095, 29.972, 54.185, -18.648]
  Call Extruder(21877.08576)
  MoveL 2296 to (23.85, 49.52, 100) mm, rotated rx -180 ry 0 rz 180 deg; joints [-154.667, -54.626, -86.349, 31.357, 55.312, -19.126]
  Call Extruder(21888.01590)
  MoveL 2297 to (12.23, 53.59, 100) mm, rotated rx 180 ry 0 rz -180 deg; joints [-153.426, -54.021, -87.94, 32.419, 56.558, -19.29]
  Call Extruder(21898.94612)
  MoveL 2298 to (0, 54.97, 100) mm, rotated rx 180 ry 0 rz 180 deg; joints [-152.438, -53.328, -89.798, 33.123, 57.863, -19.141]
  Call Extruder(21909.87635)
  MoveL 2299 to (-12.23, 53.59, 100) mm, rotated rx 180 ry 0 rz 180 deg; joints [-151.764, -52.585, -91.839, 33.434, 59.166, -18.696]
  Call Extruder(21920.80648)
  MoveL 2300 to (-23.85, 49.52, 100) mm, rotated rx -180 ry 0 rz 180 deg; joints [-151.463, -51.833, -93.968, 33.324, 60.41, -17.986]
  Call Extruder(21931.73676)
  MoveL 2301 to (-34.27, 42.98, 100) mm, rotated rx 180 ry 0 rz 180 deg; joints [-151.589, -51.109, -96.084, 32.765, 61.539, -17.052]
  Call Extruder(21942.66688)
  MoveL 2302 to (-42.98, 34.27, 100) mm, rotated rx 180 ry 0 rz -180 deg; joints [-152.179, -50.45, -98.08, 31.745, 62.503, -15.942]
  Call Extruder(21953.59716)
  MoveL 2303 to (-49.52, 23.85, 100) mm, rotated rx 180 ry 0 rz 180 deg; joints [-153.248, -49.887, -99.851, 30.269, 63.256, -14.716]
  Call Extruder(21964.52730)
  MoveL 2304 to (-53.59, 12.23, 100) mm, rotated rx 180 ry 0 rz 180 deg; joints [-154.769, -49.445, -101.294, 28.375, 63.759, -13.432]
  Call Extruder(21975.45752)
  MoveL 2305 to (-54.97, 0, 100) mm, rotated rx 180 ry 0 rz -180 deg; joints [-156.673, -49.14, -102.322, 26.145, 63.979, -12.153]
  Call Extruder(21980.98314)
  MoveL 2306 to (-54.27, -6.18, 100) mm, rotated rx 180 ry 0 rz 180 deg; joints [-157.76, -49.057, -102.607, 24.918, 63.938, -11.536]
  Set speed (130.0 mm/s)
  MoveL 2307 to (-49.9, -9.51, 100) mm, rotated rx -180 ry 0 rz 180 deg; joints [-158.616, -49.191, -102.147, 24.049, 63.473, -11.271]
  MoveL 2308 to (2.94, -13, 100) mm, rotated rx 180 ry 0 rz 180 deg; joints [-162.152, -51.833, -93.967, 21.272, 57.654, -11.766]
  Call Extruder(21985.68214)
  Set speed (80.0 mm/s)
  MoveL 2309 to (5.78, -12.01, 100) mm, rotated rx 180 ry 0 rz 180 deg; joints [-162.141, -52.016, -93.444, 21.364, 57.339, -11.92]
  Call Extruder(21990.34576)
  MoveL 2310 to (8.31, -10.42, 100) mm, rotated rx -180 ry 0 rz -180 deg; joints [-162.027, -52.194, -92.938, 21.573, 57.058, -12.134]
  Call Extruder(21995.00995)
  MoveL 2311 to (10.42, -8.31, 100) mm, rotated rx 180 ry 0 rz 180 deg; joints [-161.819, -52.359, -92.471, 21.888, 56.822, -12.4]
  Call Extruder(21999.67358)
  MoveL 2312 to (12.01, -5.78, 100) mm, rotated rx 180 ry 0 rz 180 deg; joints [-161.529, -52.504, -92.066, 22.291, 56.644, -12.703]
  Call Extruder(22004.33714)
  MoveL 2313 to (13, -2.97, 100) mm, rotated rx 180 ry 0 rz -180 deg; joints [-161.171, -52.62, -91.742, 22.762, 56.531, -13.028]
  Call Extruder(22009.00110)
  MoveL 2314 to (13.33, 0, 100) mm, rotated rx 180 ry 0 rz 180 deg; joints [-160.763, -52.702, -91.515, 23.276, 56.491, -13.359]
  Call Extruder(22013.66505)
  MoveL 2315 to (13, 2.97, 100) mm, rotated rx 180 ry 0 rz 180 deg; joints [-160.324, -52.745, -91.395, 23.808, 56.524, -13.678]
  Call Extruder(22018.32863)
  MoveL 2316 to (12.01, 5.78, 100) mm, rotated rx 180 ry 0 rz -180 deg; joints [-159.874, -52.747, -91.39, 24.332, 56.628, -13.968]
  Call Extruder(22022.99225)
  MoveL 2317 to (10.42, 8.31, 100) mm, rotated rx 180 ry 0 rz 180 deg; joints [-159.432, -52.708, -91.498, 24.825, 56.798, -14.215]
  Call Extruder(22027.65644)
  MoveL 2318 to (8.31, 10.42, 100) mm, rotated rx -180 ry 0 rz -180 deg; joints [-159.021, -52.63, -91.715, 25.263, 57.025, -14.405]
  Call Extruder(22032.32007)
  MoveL 2319 to (5.78, 12.01, 100) mm, rotated rx 180 ry 0 rz 180 deg; joints [-158.657, -52.517, -92.03, 25.626, 57.299, -14.529]
  Call Extruder(22036.98364)
  MoveL 2320 to (2.97, 13, 100) mm, rotated rx -180 ry 0 rz 180 deg; joints [-158.359, -52.375, -92.428, 25.897, 57.604, -14.581]
  Call Extruder(22041.64760)
  MoveL 2321 to (0, 13.33, 100) mm, rotated rx -180 ry 0 rz 180 deg; joints [-158.143, -52.211, -92.89, 26.063, 57.926, -14.559]
  Call Extruder(22046.31155)
  MoveL 2322 to (-2.97, 13, 100) mm, rotated rx -180 ry 0 rz -180 deg; joints [-158.019, -52.034, -93.392, 26.115, 58.25, -14.465]
  Call Extruder(22050.97511)
  MoveL 2323 to (-5.78, 12.01, 100) mm, rotated rx 180 ry 0 rz 180 deg; joints [-157.997, -51.852, -93.912, 26.048, 58.558, -14.303]
  Call Extruder(22055.63875)
  MoveL 2324 to (-8.31, 10.42, 100) mm, rotated rx 180 ry 0 rz 180 deg; joints [-158.08, -51.675, -94.421, 25.866, 58.837, -14.084]
  Call Extruder(22060.30294)
  MoveL 2325 to (-10.42, 8.31, 100) mm, rotated rx 180 ry 0 rz 180 deg; joints [-158.266, -51.512, -94.895, 25.573, 59.072, -13.818]
  Call Extruder(22064.96656)
  MoveL 2326 to (-12.01, 5.78, 100) mm, rotated rx 180 ry 0 rz -180 deg; joints [-158.549, -51.371, -95.309, 25.184, 59.252, -13.518]
  Call Extruder(22069.63013)
  MoveL 2327 to (-12.99, 2.97, 100) mm, rotated rx 180 ry 0 rz -180 deg; joints [-158.913, -51.257, -95.643, 24.717, 59.367, -13.2]
  Call Extruder(22074.29409)
  MoveL 2328 to (-13.33, 0, 100) mm, rotated rx -180 ry 0 rz 180 deg; joints [-159.341, -51.178, -95.877, 24.194, 59.412, -12.878]
  Call Extruder(22078.95804)
  MoveL 2329 to (-12.99, -2.97, 100) mm, rotated rx 180 ry 0 rz -180 deg; joints [-159.811, -51.137, -96, 23.643, 59.383, -12.569]
  Call Extruder(22083.62161)
  MoveL 2330 to (-12.01, -5.78, 100) mm, rotated rx 180 ry 0 rz -180 deg; joints [-160.294, -51.135, -96.006, 23.092, 59.283, -12.287]
  Call Extruder(22088.28524)
  MoveL 2331 to (-10.42, -8.31, 100) mm, rotated rx 180 ry 0 rz 180 deg; joints [-160.766, -51.172, -95.894, 22.572, 59.115, -12.045]
  Call Extruder(22092.94943)
  MoveL 2332 to (-8.31, -10.42, 100) mm, rotated rx 180 ry 0 rz 180 deg; joints [-161.2, -51.248, -95.671, 22.112, 58.888, -11.856]
  Call Extruder(22097.61305)
  MoveL 2333 to (-5.78, -12.01, 100) mm, rotated rx 180 ry 0 rz 180 deg; joints [-161.572, -51.358, -95.346, 21.734, 58.614, -11.729]
  Call Extruder(22102.27662)
  MoveL 2334 to (-2.97, -13, 100) mm, rotated rx -180 ry 0 rz 180 deg; joints [-161.863, -51.497, -94.939, 21.461, 58.305, -11.67]
  Call Extruder(22106.94058)
  MoveL 2335 to (0, -13.33, 100) mm, rotated rx -180 ry 0 rz -180 deg; joints [-162.059, -51.658, -94.47, 21.304, 57.979, -11.683]
  Call Extruder(22111.56821)
  MoveL 2336 to (2.94, -13, 100) mm, rotated rx 180 ry 0 rz 180 deg; joints [-162.152, -51.833, -93.967, 21.272, 57.654, -11.766]
  Set speed (130.0 mm/s)
  MoveL 2337 to (2.94, -13, 105) mm, rotated rx 180 ry 0 rz 180 deg; joints [-162.152, -51.073, -94.278, 21.376, 57.235, -11.96]
  MoveL 2338 to (-26.25, -4.54, 105) mm, rotated rx 180 ry 0 rz 180 deg; joints [-159.288, -49.618, -98.518, 23.998, 60.41, -12.398]
  Call Extruder(22113.80083)
  Set speed (60.0 mm/s)
  MoveL 2339 to (-26.09, -5.96, 105) mm, rotated rx 180 ry 0 rz 180 deg; joints [-159.522, -49.598, -98.577, 23.727, 60.396, -12.25]
  Call Extruder(22123.16562)
  MoveL 2340 to (-24.11, -11.61, 105) mm, rotated rx 180 ry 0 rz 180 deg; joints [-160.532, -49.594, -98.589, 22.588, 60.194, -11.683]
  Call Extruder(22132.53054)
  MoveL 2341 to (-20.93, -16.69, 105) mm, rotated rx 180 ry 0 rz 180 deg; joints [-161.513, -49.67, -98.359, 21.51, 59.857, -11.195]
  Call Extruder(22141.89574)
  MoveL 2342 to (-16.69, -20.93, 105) mm, rotated rx -180 ry 0 rz -180 deg; joints [-162.406, -49.823, -97.9, 20.559, 59.401, -10.808]
  Call Extruder(22151.26067)
  MoveL 2343 to (-11.61, -24.12, 105) mm, rotated rx -180 ry 0 rz 180 deg; joints [-163.159, -50.046, -97.238, 19.787, 58.849, -10.542]
  Call Extruder(22160.62546)
  MoveL 2344 to (-5.96, -26.09, 105) mm, rotated rx -180 ry 0 rz 180 deg; joints [-163.733, -50.329, -96.409, 19.237, 58.229, -10.411]
  Call Extruder(22169.99056)
  MoveL 2345 to (0, -26.77, 105) mm, rotated rx -180 ry 0 rz 180 deg; joints [-164.103, -50.658, -95.458, 18.935, 57.575, -10.423]
  Call Extruder(22177.62497)
  MoveL 2346 to (4.86, -26.22, 105) mm, rotated rx -180 ry 0 rz 180 deg; joints [-164.23, -50.95, -94.624, 18.9, 57.04, -10.552]
  Call Extruder(22179.35567)
  MoveL 2347 to (5.96, -26.09, 105) mm, rotated rx 180 ry 0 rz 180 deg; joints [-164.258, -51.017, -94.434, 18.893, 56.919, -10.581]
  Call Extruder(22188.72047)
  MoveL 2348 to (11.61, -24.11, 105) mm, rotated rx 180 ry 0 rz 180 deg; joints [-164.201, -51.39, -93.391, 19.104, 56.294, -10.88]
  Call Extruder(22198.08538)
  MoveL 2349 to (16.69, -20.93, 105) mm, rotated rx -180 ry 0 rz 180 deg; joints [-163.944, -51.756, -92.379, 19.552, 55.734, -11.308]
  Call Extruder(22207.45059)
  MoveL 2350 to (20.93, -16.69, 105) mm, rotated rx -180 ry 0 rz 180 deg; joints [-163.508, -52.097, -91.447, 20.208, 55.267, -11.845]
  Call Extruder(22216.81551)
  MoveL 2351 to (24.11, -11.61, 105) mm, rotated rx -180 ry 0 rz 180 deg; joints [-162.92, -52.396, -90.64, 21.034, 54.916, -12.464]
  Call Extruder(22226.18030)
  MoveL 2352 to (26.09, -5.96, 105) mm, rotated rx -180 ry 0 rz -180 deg; joints [-162.209, -52.637, -89.997, 21.986, 54.698, -13.133]
  Call Extruder(22235.54540)
  MoveL 2353 to (26.77, 0, 105) mm, rotated rx -180 ry 0 rz -180 deg; joints [-161.41, -52.806, -89.547, 23.015, 54.625, -13.816]
  Call Extruder(22244.91051)
  MoveL 2354 to (26.09, 5.96, 105) mm, rotated rx -180 ry 0 rz 180 deg; joints [-160.556, -52.895, -89.311, 24.072, 54.699, -14.475]
  Call Extruder(22254.27531)
  MoveL 2355 to (24.11, 11.61, 105) mm, rotated rx 180 ry 0 rz -180 deg; joints [-159.683, -52.9, -89.299, 25.107, 54.915, -15.074]
  Call Extruder(22263.64022)
  MoveL 2356 to (20.93, 16.69, 105) mm, rotated rx 180 ry 0 rz 180 deg; joints [-158.826, -52.819, -89.514, 26.075, 55.262, -15.581]
  Call Extruder(22273.00543)
  MoveL 2357 to (16.69, 20.93, 105) mm, rotated rx -180 ry 0 rz 180 deg; joints [-158.019, -52.657, -89.943, 26.934, 55.721, -15.969]
  Call Extruder(22282.37034)
  MoveL 2358 to (11.61, 24.12, 105) mm, rotated rx 180 ry 0 rz 180 deg; joints [-157.299, -52.423, -90.569, 27.648, 56.269, -16.22]
  Call Extruder(22291.73515)
  MoveL 2359 to (5.96, 26.09, 105) mm, rotated rx 180 ry 0 rz 180 deg; joints [-156.697, -52.129, -91.361, 28.187, 56.878, -16.322]
  Call Extruder(22301.10025)
  MoveL 2360 to (0, 26.77, 105) mm, rotated rx 180 ry 0 rz 180 deg; joints [-156.245, -51.791, -92.282, 28.525, 57.518, -16.272]
  Call Extruder(22310.46535)
  MoveL 2361 to (-5.96, 26.09, 105) mm, rotated rx 180 ry 0 rz 180 deg; joints [-155.969, -51.427, -93.288, 28.644, 58.158, -16.076]
  Call Extruder(22319.83014)
  MoveL 2362 to (-11.61, 24.12, 105) mm, rotated rx 180 ry 0 rz 180 deg; joints [-155.891, -51.054, -94.331, 28.536, 58.768, -15.746]
  Call Extruder(22329.19506)
  MoveL 2363 to (-16.69, 20.93, 105) mm, rotated rx 180 ry 0 rz -180 deg; joints [-156.025, -50.692, -95.359, 28.195, 59.318, -15.299]
  Call Extruder(22338.56027)
  MoveL 2364 to (-20.93, 16.69, 105) mm, rotated rx 180 ry 0 rz 180 deg; joints [-156.374, -50.359, -96.319, 27.632, 59.782, -14.76]
  Call Extruder(22347.92518)
  MoveL 2365 to (-24.11, 11.61, 105) mm, rotated rx 180 ry 0 rz 180 deg; joints [-156.928, -50.072, -97.162, 26.865, 60.137, -14.156]
  Call Extruder(22357.28998)
  MoveL 2366 to (-26.09, 5.96, 105) mm, rotated rx 180 ry 0 rz -180 deg; joints [-157.665, -49.842, -97.843, 25.926, 60.365, -13.516]
  Call Extruder(22366.65509)
  MoveL 2367 to (-26.77, 0, 105) mm, rotated rx -180 ry 0 rz -180 deg; joints [-158.546, -49.682, -98.323, 24.861, 60.454, -12.871]
  Call Extruder(22371.44382)
  MoveL 2368 to (-26.42, -3.05, 105) mm, rotated rx -180 ry 0 rz 180 deg; joints [-159.044, -49.638, -98.455, 24.282, 60.424, -12.553]
  Set speed (130.0 mm/s)
  MoveL 2369 to (-41.86, -6.29, 105) mm, rotated rx 180 ry 0 rz 180 deg; joints [-158.606, -48.8, -101.053, 24.374, 62.121, -11.962]
  Call Extruder(22376.44167)
  Set speed (60.0 mm/s)
  MoveL 2370 to (-41.5, -9.47, 105) mm, rotated rx 180 ry 0 rz -180 deg; joints [-159.151, -48.758, -101.187, 23.749, 62.093, -11.636]
  Call Extruder(22391.33732)
  MoveL 2371 to (-38.36, -18.47, 105) mm, rotated rx 180 ry 0 rz 180 deg; joints [-160.835, -48.752, -101.207, 21.874, 61.779, -10.749]
  Call Extruder(22406.23318)
  MoveL 2372 to (-33.28, -26.54, 105) mm, rotated rx 180 ry 0 rz 180 deg; joints [-162.466, -48.87, -100.831, 20.1, 61.245, -9.984]
  Call Extruder(22421.12899)
  MoveL 2373 to (-26.54, -33.28, 105) mm, rotated rx -180 ry 0 rz -180 deg; joints [-163.93, -49.108, -100.084, 18.542, 60.518, -9.373]
  Call Extruder(22436.02484)
  MoveL 2374 to (-18.47, -38.36, 105) mm, rotated rx -180 ry 0 rz 180 deg; joints [-165.137, -49.456, -99.01, 17.295, 59.635, -8.945]
  Call Extruder(22450.92049)
  MoveL 2375 to (-9.47, -41.5, 105) mm, rotated rx 180 ry 0 rz 180 deg; joints [-166.024, -49.9, -97.672, 16.428, 58.643, -8.723]
  Call Extruder(22465.81637)
  MoveL 2376 to (0, -42.57, 105) mm, rotated rx 180 ry 0 rz 180 deg; joints [-166.562, -50.419, -96.146, 15.977, 57.595, -8.723]
  Call Extruder(22476.21632)
  MoveL 2377 to (6.61, -41.83, 105) mm, rotated rx -180 ry 0 rz 180 deg; joints [-166.691, -50.815, -95.008, 15.957, 56.862, -8.884]
  Call Extruder(22480.71224)
  MoveL 2378 to (9.47, -41.51, 105) mm, rotated rx -180 ry 0 rz 180 deg; joints [-166.745, -50.989, -94.513, 15.951, 56.545, -8.954]
  Call Extruder(22495.60790)
  MoveL 2379 to (18.47, -38.36, 105) mm, rotated rx 180 ry 0 rz 180 deg; joints [-166.591, -51.583, -92.856, 16.333, 55.547, -9.413]
  Call Extruder(22510.50375)
  MoveL 2380 to (26.54, -33.29, 105) mm, rotated rx 180 ry 0 rz -180 deg; joints [-166.133, -52.168, -91.255, 17.088, 54.653, -10.084]
  Call Extruder(22525.39957)
  MoveL 2381 to (33.29, -26.54, 105) mm, rotated rx 180 ry 0 rz 180 deg; joints [-165.409, -52.716, -89.787, 18.164, 53.908, -10.939]
  Call Extruder(22540.29542)
  MoveL 2382 to (38.36, -18.47, 105) mm, rotated rx -180 ry 0 rz 180 deg; joints [-164.468, -53.196, -88.519, 19.498, 53.349, -11.935]
  Call Extruder(22555.19107)
  MoveL 2383 to (41.5, -9.47, 105) mm, rotated rx -180 ry 0 rz -180 deg; joints [-163.355, -53.583, -87.51, 21.017, 53.006, -13.017]
  Call Extruder(22570.08694)
  MoveL 2384 to (42.57, 0, 105) mm, rotated rx 180 ry 0 rz 180 deg; joints [-162.12, -53.856, -86.804, 22.642, 52.894, -14.125]
  Call Extruder(22584.98282)
  MoveL 2385 to (41.5, 9.47, 105) mm, rotated rx 180 ry 0 rz 180 deg; joints [-160.81, -54, -86.434, 24.298, 53.018, -15.194]
  Call Extruder(22599.87848)
  MoveL 2386 to (38.36, 18.47, 105) mm, rotated rx 180 ry 0 rz 180 deg; joints [-159.475, -54.007, -86.416, 25.907, 53.369, -16.162]
  Call Extruder(22614.77432)
  MoveL 2387 to (33.29, 26.54, 105) mm, rotated rx 180 ry 0 rz -180 deg; joints [-158.16, -53.877, -86.752, 27.403, 53.927, -16.975]
  Call Extruder(22629.67015)
  MoveL 2388 to (26.54, 33.28, 105) mm, rotated rx 180 ry 0 rz 180 deg; joints [-156.916, -53.616, -87.426, 28.728, 54.661, -17.59]
  Call Extruder(22644.56599)
  MoveL 2389 to (18.47, 38.36, 105) mm, rotated rx -180 ry 0 rz -180 deg; joints [-155.789, -53.239, -88.407, 29.83, 55.533, -17.979]
  Call Extruder(22659.46165)
  MoveL 2390 to (9.47, 41.51, 105) mm, rotated rx -180 ry 0 rz 180 deg; joints [-154.828, -52.767, -89.652, 30.669, 56.498, -18.125]
  Call Extruder(22674.35753)
  MoveL 2391 to (0, 42.57, 105) mm, rotated rx 180 ry 0 rz 180 deg; joints [-154.081, -52.225, -91.103, 31.212, 57.509, -18.029]
  Call Extruder(22689.25340)
  MoveL 2392 to (-9.47, 41.51, 105) mm, rotated rx 180 ry 0 rz 180 deg; joints [-153.594, -51.642, -92.693, 31.432, 58.519, -17.701]
  Call Extruder(22704.14905)
  MoveL 2393 to (-18.47, 38.36, 105) mm, rotated rx 180 ry 0 rz 180 deg; joints [-153.408, -51.048, -94.349, 31.306, 59.481, -17.163]
  Call Extruder(22719.04490)
  MoveL 2394 to (-26.54, 33.29, 105) mm, rotated rx 180 ry 0 rz 180 deg; joints [-153.557, -50.474, -95.988, 30.824, 60.35, -16.445]
  Call Extruder(22733.94072)
  MoveL 2395 to (-33.29, 26.54, 105) mm, rotated rx 180 ry 0 rz 180 deg; joints [-154.059, -49.948, -97.528, 29.982, 61.087, -15.586]
  Call Extruder(22748.83657)
  MoveL 2396 to (-38.36, 18.47, 105) mm, rotated rx 180 ry 0 rz 180 deg; joints [-154.913, -49.496, -98.888, 28.8, 61.655, -14.629]
  Call Extruder(22763.73223)
  MoveL 2397 to (-41.51, 9.47, 105) mm, rotated rx 180 ry 0 rz -180 deg; joints [-156.091, -49.138, -99.991, 27.317, 62.025, -13.62]
  Call Extruder(22778.62810)
  MoveL 2398 to (-42.57, 0, 105) mm, rotated rx -180 ry 0 rz -180 deg; joints [-157.533, -48.888, -100.773, 25.602, 62.175, -12.607]
  Call Extruder(22786.18238)
  MoveL 2399 to (-42.03, -4.8, 105) mm, rotated rx -180 ry 0 rz 180 deg; joints [-158.35, -48.82, -100.989, 24.665, 62.134, -12.114]
  Set speed (130.0 mm/s)
  MoveL 2400 to (-54.1, -7.67, 105) mm, rotated rx 180 ry 0 rz 180 deg; joints [-158.024, -48.203, -103.002, 24.725, 63.469, -11.623]
  Call Extruder(22790.25501)
  Set speed (30.0 mm/s)
  MoveL 2401 to (-53.59, -12.23, 105) mm, rotated rx -180 ry 0 rz -180 deg; joints [-158.835, -48.144, -103.197, 23.808, 63.434, -11.163]
  Call Extruder(22801.18514)
  MoveL 2402 to (-49.52, -23.85, 105) mm, rotated rx 180 ry 0 rz 180 deg; joints [-161.095, -48.137, -103.223, 21.316, 63.035, -10.034]
  Call Extruder(22812.11543)
  MoveL 2403 to (-42.98, -34.27, 105) mm, rotated rx -180 ry 0 rz 180 deg; joints [-163.275, -48.285, -102.727, 18.959, 62.347, -9.059]
  Call Extruder(22823.04555)
  MoveL 2404 to (-34.27, -42.98, 105) mm, rotated rx -180 ry 0 rz 180 deg; joints [-165.21, -48.586, -101.742, 16.902, 61.404, -8.275]
  Call Extruder(22833.97583)
  MoveL 2405 to (-23.85, -49.53, 105) mm, rotated rx 180 ry 0 rz 180 deg; joints [-166.774, -49.028, -100.333, 15.278, 60.257, -7.718]
  Call Extruder(22844.90596)
  MoveL 2406 to (-12.23, -53.59, 105) mm, rotated rx 180 ry 0 rz 180 deg; joints [-167.889, -49.595, -98.587, 14.173, 58.97, -7.417]
  Call Extruder(22855.83619)
  MoveL 2407 to (0, -54.97, 105) mm, rotated rx 180 ry 0 rz 180 deg; joints [-168.526, -50.262, -96.604, 13.625, 57.61, -7.398]
  Call Extruder(22862.97903)
  MoveL 2408 to (7.99, -54.07, 105) mm, rotated rx 180 ry 0 rz 180 deg; joints [-168.639, -50.738, -95.227, 13.629, 56.72, -7.578]
  Call Extruder(22866.76641)
  MoveL 2409 to (12.23, -53.59, 105) mm, rotated rx 180 ry 0 rz 180 deg; joints [-168.697, -50.997, -94.491, 13.635, 56.249, -7.675]
  Call Extruder(22877.69655)
  MoveL 2410 to (23.85, -49.53, 105) mm, rotated rx 180 ry 0 rz 180 deg; joints [-168.436, -51.764, -92.356, 14.172, 54.957, -8.25]
  Call Extruder(22888.62683)
  MoveL 2411 to (34.27, -42.98, 105) mm, rotated rx 180 ry 0 rz 180 deg; joints [-167.797, -52.524, -90.3, 15.186, 53.799, -9.108]
  Call Extruder(22899.55695)
  MoveL 2412 to (42.98, -34.27, 105) mm, rotated rx 180 ry 0 rz 180 deg; joints [-166.837, -53.235, -88.417, 16.604, 52.834, -10.212]
  Call Extruder(22910.48723)
  MoveL 2413 to (49.53, -23.85, 105) mm, rotated rx 180 ry 0 rz 180 deg; joints [-165.618, -53.86, -86.795, 18.344, 52.112, -11.509]
  Call Extruder(22921.41736)
  MoveL 2414 to (53.59, -12.23, 105) mm, rotated rx 180 ry 0 rz -180 deg; joints [-164.2, -54.365, -85.503, 20.31, 51.669, -12.928]
  Call Extruder(22932.34759)
  MoveL 2415 to (54.97, 0, 105) mm, rotated rx 180 ry 0 rz 180 deg; joints [-162.641, -54.721, -84.601, 22.401, 51.529, -14.383]
  Call Extruder(22943.27781)
  MoveL 2416 to (53.59, 12.23, 105) mm, rotated rx 180 ry 0 rz 180 deg; joints [-160.996, -54.909, -84.128, 24.517, 51.695, -15.785]
  Call Extruder(22954.20795)
  MoveL 2417 to (49.52, 23.85, 105) mm, rotated rx -180 ry 0 rz -180 deg; joints [-159.322, -54.918, -84.105, 26.561, 52.156, -17.051]
  Call Extruder(22965.13823)
  MoveL 2418 to (42.98, 34.27, 105) mm, rotated rx 180 ry 0 rz 180 deg; joints [-157.673, -54.747, -84.534, 28.451, 52.884, -18.106]
  Call Extruder(22976.06835)
  MoveL 2419 to (34.27, 42.98, 105) mm, rotated rx 180 ry 0 rz 180 deg; joints [-156.102, -54.407, -85.396, 30.118, 53.837, -18.896]
  Call Extruder(22986.99863)
  MoveL 2420 to (23.85, 49.52, 105) mm, rotated rx 180 ry 0 rz 180 deg; joints [-154.667, -53.916, -86.651, 31.505, 54.963, -19.386]
  Call Extruder(22997.92877)
  MoveL 2421 to (12.23, 53.59, 105) mm, rotated rx 180 ry 0 rz 180 deg; joints [-153.426, -53.302, -88.244, 32.568, 56.207, -19.558]
  Call Extruder(23008.85899)
  MoveL 2422 to (0, 54.97, 105) mm, rotated rx -180 ry 0 rz 180 deg; joints [-152.438, -52.597, -90.104, 33.271, 57.506, -19.417]
  Call Extruder(23019.78921)
  MoveL 2423 to (-12.23, 53.59, 105) mm, rotated rx 180 ry 0 rz 180 deg; joints [-151.764, -51.841, -92.147, 33.58, 58.802, -18.978]
  Call Extruder(23030.71935)
  MoveL 2424 to (-23.85, 49.52, 105) mm, rotated rx 180 ry 0 rz 180 deg; joints [-151.463, -51.072, -94.279, 33.465, 60.035, -18.271]
  Call Extruder(23041.64963)
  MoveL 2425 to (-34.27, 42.98, 105) mm, rotated rx 180 ry 0 rz 180 deg; joints [-151.589, -50.332, -96.398, 32.902, 61.151, -17.337]
  Call Extruder(23052.57975)
  MoveL 2426 to (-42.98, 34.27, 105) mm, rotated rx 180 ry 0 rz -180 deg; joints [-152.179, -49.657, -98.399, 31.876, 62.1, -16.225]
  Call Extruder(23063.51003)
  MoveL 2427 to (-49.52, 23.85, 105) mm, rotated rx -180 ry 0 rz 180 deg; joints [-153.248, -49.079, -100.174, 30.394, 62.837, -14.991]
  Call Extruder(23074.44017)
  MoveL 2428 to (-53.59, 12.23, 105) mm, rotated rx 180 ry 0 rz 180 deg; joints [-154.769, -48.623, -101.62, 28.493, 63.323, -13.696]
  Call Extruder(23085.37039)
  MoveL 2429 to (-54.97, 0, 105) mm, rotated rx 180 ry 0 rz -180 deg; joints [-156.673, -48.308, -102.651, 26.255, 63.528, -12.4]
  Call Extruder(23090.89601)
  MoveL 2430 to (-54.27, -6.18, 105) mm, rotated rx 180 ry 0 rz 180 deg; joints [-157.76, -48.222, -102.936, 25.024, 63.481, -11.774]
  Set speed (130.0 mm/s)
  MoveL 2431 to (-49.9, -9.51, 105) mm, rotated rx 180 ry 0 rz 180 deg; joints [-158.616, -48.361, -102.476, 24.152, 63.015, -11.501]
  MoveL 2432 to (2.97, -12.99, 105) mm, rotated rx 180 ry 0 rz -180 deg; joints [-162.152, -51.074, -94.274, 21.376, 57.233, -11.961]
  Call Extruder(23095.55958)
  Set speed (80.0 mm/s)
  MoveL 2433 to (5.78, -12.01, 105) mm, rotated rx 180 ry 0 rz 180 deg; joints [-162.141, -51.259, -93.754, 21.469, 56.924, -12.114]
  Call Extruder(23100.22320)
  MoveL 2434 to (8.31, -10.42, 105) mm, rotated rx -180 ry 0 rz -180 deg; joints [-162.027, -51.441, -93.247, 21.68, 56.646, -12.329]
  Call Extruder(23104.88739)
  MoveL 2435 to (10.42, -8.31, 105) mm, rotated rx 180 ry 0 rz 180 deg; joints [-161.819, -51.61, -92.78, 21.997, 56.413, -12.597]
  Call Extruder(23109.55102)
  MoveL 2436 to (12.01, -5.78, 105) mm, rotated rx -180 ry 0 rz 180 deg; joints [-161.529, -51.758, -92.374, 22.402, 56.238, -12.903]
  Call Extruder(23114.21459)
  MoveL 2437 to (13, -2.97, 105) mm, rotated rx -180 ry 0 rz -180 deg; joints [-161.171, -51.876, -92.049, 22.875, 56.129, -13.232]
  Call Extruder(23118.87855)
  MoveL 2438 to (13.33, 0, 105) mm, rotated rx -180 ry 0 rz -180 deg; joints [-160.763, -51.959, -91.822, 23.391, 56.091, -13.566]
  Call Extruder(23123.54250)
  MoveL 2439 to (13, 2.97, 105) mm, rotated rx -180 ry 0 rz 180 deg; joints [-160.324, -52.003, -91.703, 23.925, 56.126, -13.889]
  Call Extruder(23128.20607)
  MoveL 2440 to (12.01, 5.78, 105) mm, rotated rx -180 ry 0 rz -180 deg; joints [-159.874, -52.005, -91.697, 24.451, 56.232, -14.184]
  Call Extruder(23132.86970)
  MoveL 2441 to (10.42, 8.31, 105) mm, rotated rx -180 ry 0 rz 180 deg; joints [-159.432, -51.966, -91.805, 24.946, 56.403, -14.434]
  Call Extruder(23137.53389)
  MoveL 2442 to (8.31, 10.42, 105) mm, rotated rx 180 ry 0 rz 180 deg; joints [-159.021, -51.886, -92.022, 25.385, 56.631, -14.628]
  Call Extruder(23142.19751)
  MoveL 2443 to (5.78, 12.01, 105) mm, rotated rx 180 ry 0 rz 180 deg; joints [-158.657, -51.771, -92.338, 25.749, 56.904, -14.755]
  Call Extruder(23146.86108)
  MoveL 2444 to (2.97, 12.99, 105) mm, rotated rx -180 ry 0 rz 180 deg; joints [-158.359, -51.626, -92.736, 26.021, 57.208, -14.81]
  Call Extruder(23151.52504)
  MoveL 2445 to (0, 13.33, 105) mm, rotated rx -180 ry 0 rz 180 deg; joints [-158.143, -51.459, -93.199, 26.186, 57.529, -14.789]
  Call Extruder(23156.18899)
  MoveL 2446 to (-2.97, 12.99, 105) mm, rotated rx 180 ry 0 rz 180 deg; joints [-158.019, -51.278, -93.703, 26.237, 57.85, -14.696]
  Call Extruder(23160.85256)
  MoveL 2447 to (-5.78, 12.01, 105) mm, rotated rx 180 ry 0 rz 180 deg; joints [-157.997, -51.092, -94.223, 26.17, 58.155, -14.535]
  Call Extruder(23165.51619)
  MoveL 2448 to (-8.31, 10.42, 105) mm, rotated rx -180 ry 0 rz 180 deg; joints [-158.08, -50.912, -94.733, 25.986, 58.431, -14.315]
  Call Extruder(23170.18038)
  MoveL 2449 to (-10.42, 8.31, 105) mm, rotated rx 180 ry 0 rz 180 deg; joints [-158.266, -50.745, -95.208, 25.692, 58.662, -14.048]
  Call Extruder(23174.84400)
  MoveL 2450 to (-12.01, 5.78, 105) mm, rotated rx 180 ry 0 rz -180 deg; joints [-158.549, -50.6, -95.623, 25.301, 58.839, -13.745]
  Call Extruder(23179.50757)
  MoveL 2451 to (-13, 2.97, 105) mm, rotated rx 180 ry 0 rz -180 deg; joints [-158.913, -50.484, -95.956, 24.832, 58.95, -13.424]
  Call Extruder(23184.17153)
  MoveL 2452 to (-13.33, 0, 105) mm, rotated rx 180 ry 0 rz 180 deg; joints [-159.341, -50.403, -96.191, 24.307, 58.992, -13.098]
  Call Extruder(23188.83548)
  MoveL 2453 to (-12.99, -2.97, 105) mm, rotated rx 180 ry 0 rz 180 deg; joints [-159.811, -50.361, -96.315, 23.753, 58.961, -12.785]
  Call Extruder(23193.49905)
  MoveL 2454 to (-12.01, -5.78, 105) mm, rotated rx 180 ry 0 rz 180 deg; joints [-160.294, -50.359, -96.321, 23.201, 58.859, -12.498]
  Call Extruder(23198.16268)
  MoveL 2455 to (-10.42, -8.31, 105) mm, rotated rx 180 ry 0 rz 180 deg; joints [-160.766, -50.397, -96.209, 22.679, 58.69, -12.252]
  Call Extruder(23202.82687)
  MoveL 2456 to (-8.31, -10.42, 105) mm, rotated rx 180 ry 0 rz -180 deg; joints [-161.2, -50.475, -95.984, 22.217, 58.463, -12.059]
  Call Extruder(23207.49050)
  MoveL 2457 to (-5.78, -12.01, 105) mm, rotated rx 180 ry 0 rz 180 deg; joints [-161.572, -50.587, -95.66, 21.839, 58.189, -11.928]
  Call Extruder(23212.15407)
  MoveL 2458 to (-2.97, -13, 105) mm, rotated rx 180 ry 0 rz 180 deg; joints [-161.863, -50.73, -95.252, 21.565, 57.882, -11.866]
  Call Extruder(23216.81801)
  MoveL 2459 to (0, -13.33, 105) mm, rotated rx -180 ry 0 rz -180 deg; joints [-162.059, -50.894, -94.782, 21.408, 57.558, -11.877]
  Call Extruder(23221.48198)
  MoveL 2460 to (2.97, -12.99, 105) mm, rotated rx 180 ry 0 rz -180 deg; joints [-162.152, -51.074, -94.274, 21.376, 57.233, -11.961]
  Set speed (130.0 mm/s)
  MoveL 2461 to (2.97, -12.99, 110) mm, rotated rx -180 ry 0 rz -180 deg; joints [-162.152, -50.315, -94.576, 21.484, 56.807, -12.16]
  MoveL 2462 to (-26.25, -4.54, 110) mm, rotated rx 180 ry 0 rz 180 deg; joints [-159.288, -48.824, -98.827, 24.111, 59.968, -12.626]
  Call Extruder(23223.71460)
  Set speed (60.0 mm/s)
  MoveL 2463 to (-26.09, -5.96, 110) mm, rotated rx -180 ry 0 rz 180 deg; joints [-159.522, -48.804, -98.886, 23.839, 59.953, -12.475]
  Call Extruder(23233.07938)
  MoveL 2464 to (-24.11, -11.61, 110) mm, rotated rx 180 ry 0 rz 180 deg; joints [-160.532, -48.8, -98.899, 22.696, 59.747, -11.898]
  Call Extruder(23242.44431)
  MoveL 2465 to (-20.93, -16.69, 110) mm, rotated rx -180 ry 0 rz 180 deg; joints [-161.513, -48.878, -98.668, 21.614, 59.408, -11.401]
  Call Extruder(23251.80951)
  MoveL 2466 to (-16.69, -20.93, 110) mm, rotated rx 180 ry 0 rz 180 deg; joints [-162.406, -49.035, -98.208, 20.659, 58.952, -11.005]
  Call Extruder(23261.17443)
  MoveL 2467 to (-11.61, -24.12, 110) mm, rotated rx 180 ry 0 rz 180 deg; joints [-163.159, -49.264, -97.545, 19.885, 58.401, -10.731]
  Call Extruder(23270.53922)
  MoveL 2468 to (-5.96, -26.09, 110) mm, rotated rx -180 ry 0 rz 180 deg; joints [-163.733, -49.553, -96.714, 19.334, 57.786, -10.594]
  Call Extruder(23279.90433)
  MoveL 2469 to (0, -26.77, 110) mm, rotated rx 180 ry 0 rz 180 deg; joints [-164.103, -49.89, -95.762, 19.032, 57.136, -10.602]
  Call Extruder(23288.19478)
  MoveL 2470 to (5.27, -26.17, 110) mm, rotated rx 180 ry 0 rz -180 deg; joints [-164.24, -50.215, -94.854, 18.995, 56.56, -10.741]
  Call Extruder(23289.26943)
  MoveL 2471 to (5.96, -26.09, 110) mm, rotated rx 180 ry 0 rz 180 deg; joints [-164.258, -50.257, -94.736, 18.99, 56.485, -10.759]
  Call Extruder(23298.63423)
  MoveL 2472 to (11.61, -24.11, 110) mm, rotated rx 180 ry 0 rz 180 deg; joints [-164.201, -50.637, -93.691, 19.204, 55.867, -11.059]
  Call Extruder(23307.99914)
  MoveL 2473 to (16.69, -20.93, 110) mm, rotated rx 180 ry 0 rz 180 deg; joints [-163.944, -51.011, -92.677, 19.655, 55.314, -11.489]
  Call Extruder(23317.36435)
  MoveL 2474 to (20.93, -16.69, 110) mm, rotated rx 180 ry 0 rz 180 deg; joints [-163.508, -51.359, -91.744, 20.315, 54.853, -12.031]
  Call Extruder(23326.72927)
  MoveL 2475 to (24.12, -11.61, 110) mm, rotated rx 180 ry 0 rz 180 deg; joints [-162.92, -51.663, -90.937, 21.146, 54.508, -12.656]
  Call Extruder(23336.09406)
  MoveL 2476 to (26.09, -5.96, 110) mm, rotated rx 180 ry 0 rz -180 deg; joints [-162.209, -51.908, -90.293, 22.102, 54.297, -13.333]
  Call Extruder(23345.45917)
  MoveL 2477 to (26.77, 0, 110) mm, rotated rx -180 ry 0 rz -180 deg; joints [-161.41, -52.08, -89.842, 23.136, 54.229, -14.023]
  Call Extruder(23354.82427)
  MoveL 2478 to (26.09, 5.96, 110) mm, rotated rx -180 ry 0 rz 180 deg; joints [-160.556, -52.171, -89.606, 24.197, 54.307, -14.691]
  Call Extruder(23364.18907)
  MoveL 2479 to (24.11, 11.61, 110) mm, rotated rx 180 ry 0 rz 180 deg; joints [-159.683, -52.176, -89.594, 25.236, 54.527, -15.298]
  Call Extruder(23373.55399)
  MoveL 2480 to (20.93, 16.69, 110) mm, rotated rx 180 ry 0 rz 180 deg; joints [-158.826, -52.093, -89.809, 26.208, 54.876, -15.812]
  Call Extruder(23382.91920)
  MoveL 2481 to (16.69, 20.93, 110) mm, rotated rx 180 ry 0 rz 180 deg; joints [-158.019, -51.929, -90.239, 27.069, 55.336, -16.208]
  Call Extruder(23392.28411)
  MoveL 2482 to (11.61, 24.12, 110) mm, rotated rx 180 ry 0 rz 180 deg; joints [-157.299, -51.691, -90.865, 27.785, 55.883, -16.464]
  Call Extruder(23401.64891)
